	W =    40.518 deg,	P =    40.131 deg,	R =    79.815 deg
   GP2:
	UF : 1, UT : 1,
	J1=    80.000 deg,	J2=    90.000 deg
};
P[269]{
   GP1:
	UF : 1, UT : 1,		CONFIG : 'N U T, 0, 0, 0',
	X =  1902.999  mm,	Y =   -46.261  mm,	Z =   175.051  mm,
	W =    52.365 deg,	P =    -4.474 deg,	R =   -14.021 deg
   GP2:
	UF : 1, UT : 1,
	J1=    90.000 deg,	J2=    90.000 deg
};
P[270]{
   GP1:
	UF : 1, UT : 1,		CONFIG : 'N U T, 0, 0, 0',
	X =  1161.856  mm,	Y =   -92.689  mm,	Z =   175.051  mm,
	W =    38.130 deg,	P =    -5.720 deg,	R =    -4.359 deg
   GP2:
	UF : 1, UT : 1,
	J1=    90.000 deg,	J2=    90.000 deg
};
P[271]{
   GP1:
	UF : 1, UT : 1,		CONFIG : 'N U T, 0, 0, 0',
	X =  1353.427  mm,	Y =   457.025  mm,	Z =   417.051  mm,
	W =    -2.563 deg,	P =     5.520 deg,	R =     2.347 deg
   GP2:
	UF : 1, UT : 1,
	J1=    90.000 deg,	J2=    90.000 deg
};
P[272]{
   GP1:
	UF : 1, UT : 1,		CONFIG : 'N U T, 0, 0, 0',
	X =  1530.428  mm,	Y =   623.025  mm,	Z =   175.051  mm,
	W =   -41.304 deg,	P =     5.776 deg,	R =    -1.616 deg
   GP2:
	UF : 1, UT : 1,
	J1=    90.000 deg,	J2=    90.000 deg
};
P[273]{
   GP1:
	UF : 1, UT : 1,		CONFIG : 'N U T, 0, 0, 0',
	X =  2221.857  mm,	Y =   134.025  mm,	Z =   133.501  mm,
	W =   -39.814 deg,	P =   -13.337 deg,	R =   -23.619 deg
   GP2:
	UF : 1, UT : 1,
	J1=    90.000 deg,	J2=    90.000 deg
};
P[274]{
   GP1:
	UF : 1, UT : 1,		CONFIG : 'N U T, 0, 0, 0',
	X =  1662.172  mm,	Y =  -195.303  mm,	Z =   -14.365  mm,
	W =    38.570 deg,	P =    15.648 deg,	R =    22.724 deg
   GP2:
	UF : 1, UT : 1,
	J1=    90.000 deg,	J2=    90.000 deg
};
P[275]{
   GP1:
	UF : 1, UT : 1,		CONFIG : 'N U T, 0, 0, 0',
	X =  1700.747  mm,	Y =  -196.414  mm,	Z =   -14.295  mm,
	W =    38.571 deg,	P =    15.644 deg,	R =   -27.579 deg
   GP2:
	UF : 1, UT : 1,
	J1=    90.000 deg,	J2=    90.000 deg
};
P[276]{
   GP1:
	UF : 1, UT : 1,		CONFIG : 'N U T, 0, 0, 0',
	X =  2162.665  mm,	Y =   110.242  mm,	Z =    59.358  mm,
	W =   -44.607 deg,	P =    -6.682 deg,	R =    -6.729 deg
   GP2:
	UF : 1, UT : 1,
	J1=    90.000 deg,	J2=    90.000 deg
};
P[277]{
   GP1:
	UF : 1, UT : 1,		CONFIG : 'N U T, 0, 0, 0',
	X =  1967.532  mm,	Y =  -196.842  mm,	Z =   -17.295  mm,
	W =    38.571 deg,	P =    15.644 deg,	R =   -27.579 deg
   GP2:
	UF : 1, UT : 1,
	J1=    90.000 deg,	J2=    90.000 deg
};
P[278]{
   GP1:
	UF : 1, UT : 1,		CONFIG : 'N U T, 0, 0, 0',
	X =  1986.786  mm,	Y =  -196.805  mm,	Z =   -16.016  mm,
	W =    40.162 deg,	P =    14.985 deg,	R =   -66.520 deg
   GP2:
	UF : 1, UT : 1,
	J1=    89.996 deg,	J2=    90.000 deg
};
P[279]{
   GP1:
	UF : 1, UT : 1,		CONFIG : 'N U T, 0, 0, 0',
	X =  2220.705  mm,	Y =    45.955  mm,	Z =    -6.075  mm,
	W =    44.920 deg,	P =     3.025 deg,	R =    -3.029 deg
   GP2:
	UF : 1, UT : 1,
	J1=    90.000 deg,	J2=    90.000 deg
};
P[280]{
   GP1:
	UF : 1, UT : 1,		CONFIG : 'N U T, 0, 0, 0',
	X =  2200.817  mm,	Y =   103.879  mm,	Z =    45.598  mm,
	W =   -44.607 deg,	P =    -6.682 deg,	R =    -6.729 deg
   GP2:
	UF : 1, UT : 1,
	J1=    90.000 deg,	J2=    90.000 deg
};
P[281]{
   GP1:
	UF : 1, UT : 1,		CONFIG : 'N U T, 0, 0, 0',
	X =  1991.025  mm,	Y =   103.879  mm,	Z =    45.598  mm,
	W =   -44.607 deg,	P =    -6.682 deg,	R =    -6.729 deg
   GP2:
	UF : 1, UT : 1,
	J1=    90.000 deg,	J2=    90.000 deg
};
P[282]{
   GP1:
	UF : 1, UT : 1,		CONFIG : 'N U T, 0, 0, 0',
	X =  2256.491  mm,	Y =    45.955  mm,	Z =    -6.075  mm,
	W =    44.920 deg,	P =     3.025 deg,	R =    -3.029 deg
   GP2:
	UF : 1, UT : 1,
	J1=    90.000 deg,	J2=    90.000 deg
};
P[283]{
   GP1:
	UF : 1, UT : 1,		CONFIG : 'N U T, 0, 0, 0',
	X =  2146.075  mm,	Y =    43.814  mm,	Z =   -11.025  mm,
	W =    44.920 deg,	P =     3.025 deg,	R =    -3.029 deg
   GP2:
	UF : 1, UT : 1,
	J1=    90.000 deg,	J2=    90.000 deg
};
P[284]{
   GP1:
	UF : 1, UT : 1,		CONFIG : 'N U T, 0, 0, 0',
	X =  2199.218  mm,	Y =    43.814  mm,	Z =   -11.025  mm,
	W =    44.920 deg,	P =     3.025 deg,	R =    -3.029 deg
   GP2:
	UF : 1, UT : 1,
	J1=    90.000 deg,	J2=    90.000 deg
};
P[285]{
   GP1:
	UF : 1, UT : 1,		CONFIG : 'N U T, 0, 0, 0',
	X =  2086.451  mm,	Y =   114.405  mm,	Z =   133.369  mm,
	W =   -44.606 deg,	P =    -6.682 deg,	R =     6.426 deg
   GP2:
	UF : 1, UT : 1,
	J1=    90.000 deg,	J2=    90.000 deg
};
P[286]{
   GP1:
	UF : 1, UT : 1,		CONFIG : 'N U T, 0, 0, 0',
	X =  2121.394  mm,	Y =   114.404  mm,	Z =   147.283  mm,
	W =   -41.424 deg,	P =   -19.434 deg,	R =   -97.506 deg
   GP2:
	UF : 1, UT : 1,
	J1=    90.000 deg,	J2=   100.000 deg
};
P[287]{
   GP1:
	UF : 1, UT : 1,		CONFIG : 'N U T, 0, 0, 0',
	X =  2080.531  mm,	Y =    -7.596  mm,	Z =    92.282  mm,
	W =   -41.424 deg,	P =   -19.434 deg,	R =   -97.506 deg
   GP2:
	UF : 1, UT : 1,
	J1=    90.000 deg,	J2=   100.000 deg
};
P[288]{
   GP1:
	UF : 1, UT : 1,		CONFIG : 'N U T, 0, 0, 0',
	X =  2206.218  mm,	Y =    43.813  mm,	Z =   -11.025  mm,
	W =    44.920 deg,	P =     3.025 deg,	R =   -14.671 deg
   GP2:
	UF : 1, UT : 1,
	J1=    90.000 deg,	J2=    90.000 deg
};
P[289]{
   GP1:
	UF : 1, UT : 1,		CONFIG : 'N U T, 0, 0, 0',
	X =  2110.963  mm,	Y =    44.118  mm,	Z =   -20.037  mm,
	W =    44.927 deg,	P =     3.029 deg,	R =     5.583 deg
   GP2:
	UF : 1, UT : 1,
	J1=    90.000 deg,	J2=    90.000 deg
};
P[290]{
   GP1:
	UF : 1, UT : 1,		CONFIG : 'N U T, 0, 0, 0',
	X =  2080.530  mm,	Y =    -7.596  mm,	Z =    92.282  mm,
	W =   -41.424 deg,	P =   -19.434 deg,	R =   -97.506 deg
   GP2:
	UF : 1, UT : 1,
	J1=    90.000 deg,	J2=   100.000 deg
};
P[291]{
   GP1:
	UF : 1, UT : 1,		CONFIG : 'N U T, 0, 0, 0',
	X =  2080.530  mm,	Y =   309.547  mm,	Z =   503.711  mm,
	W =    -3.830 deg,	P =   -10.878 deg,	R =   -17.892 deg
   GP2:
	UF : 1, UT : 1,
	J1=    90.000 deg,	J2=   135.000 deg
};
P[292]{
   GP1:
	UF : 1, UT : 1,		CONFIG : 'N U T, 0, 0, 0',
	X =  2670.559  mm,	Y =   209.547  mm,	Z =   314.711  mm,
	W =    -3.830 deg,	P =   -10.878 deg,	R =   -17.892 deg
   GP2:
	UF : 1, UT : 1,
	J1=    90.000 deg,	J2=   135.000 deg
};
P[293]{
   GP1:
	UF : 1, UT : 1,		CONFIG : 'N U T, 0, 0, 0',
	X =  2021.034  mm,	Y =    44.118  mm,	Z =   -20.036  mm,
	W =    44.927 deg,	P =     3.029 deg,	R =     5.583 deg
   GP2:
	UF : 1, UT : 1,
	J1=    90.000 deg,	J2=    90.000 deg
};
P[294]{
   GP1:
	UF : 1, UT : 1,		CONFIG : 'N U T, 0, 0, 0',
	X =  2006.091  mm,	Y =    44.761  mm,	Z =   -20.036  mm,
	W =    44.926 deg,	P =     3.029 deg,	R =    37.260 deg
   GP2:
	UF : 1, UT : 1,
	J1=    90.000 deg,	J2=    90.000 deg
};
P[295]{
   GP1:
	UF : 1, UT : 1,		CONFIG : 'N U T, 0, 0, 0',
	X =  2649.168  mm,	Y =   166.049  mm,	Z =   301.659  mm,
	W =    13.374 deg,	P =   -35.036 deg,	R =   -22.495 deg
   GP2:
	UF : 1, UT : 1,
	J1=    90.000 deg,	J2=   135.000 deg
};
P[296]{
   GP1:
	UF : 1, UT : 1,		CONFIG : 'N U T, 0, 0, 0',
	X =  2349.168  mm,	Y =   281.049  mm,	Z =   301.659  mm,
	W =     -.090 deg,	P =    -5.498 deg,	R =      .950 deg
   GP2:
	UF : 1, UT : 1,
	J1=    90.000 deg,	J2=   135.000 deg
};
P[297]{
   GP1:
	UF : 1, UT : 1,		CONFIG : 'N U T, 0, 0, 0',
	X =  1789.966  mm,	Y =    44.323  mm,	Z =    52.714  mm,
	W =    50.325 deg,	P =     2.535 deg,	R =    12.049 deg
   GP2:
	UF : 1, UT : 1,
	J1=    90.000 deg,	J2=    90.000 deg
};
P[298]{
   GP1:
	UF : 1, UT : 1,		CONFIG : 'N U T, 0, 0, 0',
	X =  1683.323  mm,	Y =    44.322  mm,	Z =    52.714  mm,
	W =    50.813 deg,	P =     2.431 deg,	R =    12.070 deg
   GP2:
	UF : 1, UT : 1,
	J1=    90.000 deg,	J2=    90.000 deg
};
P[299]{
   GP1:
	UF : 1, UT : 1,		CONFIG : 'N U T, 0, 0, 0',
	X =  2703.820  mm,	Y =   252.204  mm,	Z =   224.219  mm,
	W =     -.140 deg,	P =    -8.465 deg,	R =      .956 deg
   GP2:
	UF : 1, UT : 1,
	J1=    90.000 deg,	J2=   135.000 deg
};
P[300]{
   GP1:
	UF : 1, UT : 1,		CONFIG : 'N U T, 0, 0, 0',
	X =  2289.178  mm,	Y =   268.490  mm,	Z =   224.220  mm,
	W =     -.140 deg,	P =    -8.465 deg,	R =      .956 deg
   GP2:
	UF : 1, UT : 1,
	J1=    90.000 deg,	J2=   135.000 deg
};
P[301]{
   GP1:
	UF : 1, UT : 1,		CONFIG : 'N U T, 0, 0, 0',
	X =  1843.464  mm,	Y =   431.347  mm,	Z =   609.934  mm,
	W =     -.140 deg,	P =    -8.465 deg,	R =   -19.002 deg
   GP2:
	UF : 1, UT : 1,
	J1=    90.000 deg,	J2=   135.000 deg
};
P[302]{
   GP1:
	UF : 1, UT : 1,		CONFIG : 'N U T, 0, 0, 0',
	X =  1843.464  mm,	Y =   431.347  mm,	Z =   378.506  mm,
	W =    39.110 deg,	P =     2.688 deg,	R =   -82.797 deg
   GP2:
	UF : 1, UT : 1,
	J1=    90.000 deg,	J2=    90.000 deg
};
P[303]{
   GP1:
	UF : 1, UT : 1,		CONFIG : 'N U T, 0, 0, 0',
	X =  2020.464  mm,	Y =   107.456  mm,	Z =   101.505  mm,
	W =    39.110 deg,	P =     2.688 deg,	R =   -82.797 deg
   GP2:
	UF : 1, UT : 1,
	J1=    90.000 deg,	J2=    90.000 deg
};
P[304]{
   GP1:
	UF : 1, UT : 1,		CONFIG : 'N U T, 0, 0, 0',
	X =  1667.771  mm,	Y =    42.806  mm,	Z =    54.038  mm,
	W =    53.172 deg,	P =     1.611 deg,	R =    24.177 deg
   GP2:
	UF : 1, UT : 1,
	J1=    90.000 deg,	J2=    90.000 deg
};
P[305]{
   GP1:
	UF : 1, UT : 1,		CONFIG : 'N U T, 0, 0, 0',
	X =  1826.870  mm,	Y =    43.892  mm,	Z =    52.359  mm,
	W =    53.726 deg,	P =    -4.474 deg,	R =     3.443 deg
   GP2:
	UF : 1, UT : 1,
	J1=    90.000 deg,	J2=    90.000 deg
};
P[306]{
   GP1:
	UF : 1, UT : 1,		CONFIG : 'N U T, 0, 0, 0',
	X =  1963.585  mm,	Y =    45.392  mm,	Z =    50.646  mm,
	W =    53.726 deg,	P =    -4.474 deg,	R =     3.443 deg
   GP2:
	UF : 1, UT : 1,
	J1=    90.000 deg,	J2=    90.000 deg
};
P[307]{
   GP1:
	UF : 1, UT : 1,		CONFIG : 'N U T, 0, 0, -1',
	X =  2012.815  mm,	Y =   114.104  mm,	Z =    90.700  mm,
	W =    40.362 deg,	P =    21.867 deg,	R =  -139.995 deg
   GP2:
	UF : 1, UT : 1,
	J1=    90.000 deg,	J2=    90.000 deg
};
P[308]{
   GP1:
	UF : 1, UT : 1,		CONFIG : 'N U T, 0, 0, 0',
	X =  1644.243  mm,	Y =   456.961  mm,	Z =    90.700  mm,
	W =   -42.959 deg,	P =    14.926 deg,	R =    16.534 deg
   GP2:
	UF : 1, UT : 1,
	J1=    90.000 deg,	J2=    90.000 deg
};
P[309]{
   GP1:
	UF : 1, UT : 1,		CONFIG : 'N U T, 0, 0, 0',
	X =  1667.302  mm,	Y =   122.961  mm,	Z =    90.700  mm,
	W =   -42.959 deg,	P =    14.926 deg,	R =    16.534 deg
   GP2:
	UF : 1, UT : 1,
	J1=    90.000 deg,	J2=    90.000 deg
};
P[310]{
   GP1:
	UF : 1, UT : 1,		CONFIG : 'N U T, 0, 0, 0',
	X =  1987.759  mm,	Y =    40.243  mm,	Z =    54.128  mm,
	W =    53.726 deg,	P =    -4.474 deg,	R =   -26.684 deg
   GP2:
	UF : 1, UT : 1,
	J1=    90.000 deg,	J2=    90.000 deg
};
P[311]{
   GP1:
	UF : 1, UT : 1,		CONFIG : 'N U T, 0, 0, 0',
	X =  2224.159  mm,	Y =    58.556  mm,	Z =    -5.448  mm,
	W =   -44.607 deg,	P =    -6.682 deg,	R =    -6.729 deg
   GP2:
	UF : 1, UT : 1,
	J1=    90.000 deg,	J2=    90.000 deg
};
P[312]{
   GP1:
	UF : 1, UT : 1,		CONFIG : 'N U T, 0, 0, 0',
	X =  2258.659  mm,	Y =    57.913  mm,	Z =    -5.448  mm,
	W =   -44.607 deg,	P =    -6.682 deg,	R =    -6.729 deg
   GP2:
	UF : 1, UT : 1,
	J1=    90.000 deg,	J2=    90.000 deg
};
P[313]{
   GP1:
	UF : 1, UT : 1,		CONFIG : 'N U T, 0, 0, 0',
	X =  2132.012  mm,	Y =    56.491  mm,	Z =   -12.327  mm,
	W =   -44.606 deg,	P =    -6.681 deg,	R =    -6.729 deg
   GP2:
	UF : 1, UT : 1,
	J1=    90.000 deg,	J2=    90.000 deg
};
P[314]{
   GP1:
	UF : 1, UT : 1,		CONFIG : 'N U T, 0, 0, 0',
	X =  2200.013  mm,	Y =    57.134  mm,	Z =   -12.327  mm,
	W =   -44.606 deg,	P =    -6.681 deg,	R =    -6.729 deg
   GP2:
	UF : 1, UT : 1,
	J1=    90.000 deg,	J2=    90.000 deg
};
P[315]{
   GP1:
	UF : 1, UT : 1,		CONFIG : 'N U T, 0, 0, 0',
	X =  2209.513  mm,	Y =    57.348  mm,	Z =   -12.326  mm,
	W =   -44.606 deg,	P =    -6.681 deg,	R =     3.931 deg
   GP2:
	UF : 1, UT : 1,
	J1=    90.000 deg,	J2=    90.000 deg
};
P[316]{
   GP1:
	UF : 1, UT : 1,		CONFIG : 'N U T, 0, 0, 0',
	X =  1985.356  mm,	Y =    56.787  mm,	Z =   -20.825  mm,
	W =   -44.607 deg,	P =    -6.682 deg,	R =    -3.024 deg
   GP2:
	UF : 1, UT : 1,
	J1=    90.000 deg,	J2=    90.000 deg
};
P[317]{
   GP1:
	UF : 1, UT : 1,		CONFIG : 'N U T, 0, 0, 0',
	X =  2092.498  mm,	Y =    57.858  mm,	Z =   -20.825  mm,
	W =   -44.607 deg,	P =    -6.682 deg,	R =    -3.024 deg
   GP2:
	UF : 1, UT : 1,
	J1=    90.000 deg,	J2=    90.000 deg
};
P[318]{
   GP1:
	UF : 1, UT : 1,		CONFIG : 'N U T, 0, 0, 0',
	X =  2108.090  mm,	Y =    59.550  mm,	Z =   -18.097  mm,
	W =   -41.242 deg,	P =   -19.883 deg,	R =    20.906 deg
   GP2:
	UF : 1, UT : 1,
	J1=    90.000 deg,	J2=    90.000 deg
};
P[319]{
   GP1:
	UF : 1, UT : 1,		CONFIG : 'N U T, 0, 0, 0',
	X =  2003.979  mm,	Y =    88.747  mm,	Z =   -10.736  mm,
	W =   -45.251 deg,	P =    -8.450 deg,	R =  -108.138 deg
   GP2:
	UF : 1, UT : 1,
	J1=    90.000 deg,	J2=   100.000 deg
};
P[320]{
   GP1:
	UF : 1, UT : 1,		CONFIG : 'N U T, 0, 0, 0',
	X =  2002.512  mm,	Y =  -133.508  mm,	Z =   -48.404  mm,
	W =   -45.251 deg,	P =    -8.450 deg,	R =   -86.327 deg
   GP2:
	UF : 1, UT : 1,
	J1=    90.000 deg,	J2=   100.000 deg
};
P[321]{
   GP1:
	UF : 1, UT : 1,		CONFIG : 'N U T, 0, 0, 0',
	X =  1385.322  mm,	Y =    99.987  mm,	Z =    81.524  mm,
	W =   -41.156 deg,	P =    19.919 deg,	R =    36.091 deg
   GP2:
	UF : 1, UT : 1,
	J1=    90.000 deg,	J2=    90.000 deg
};
P[322]{
   GP1:
	UF : 1, UT : 1,		CONFIG : 'N U T, 0, 0, 0',
	X =  1287.575  mm,	Y =   726.729  mm,	Z =   436.468  mm,
	W =   -45.215 deg,	P =    11.103 deg,	R =    59.860 deg
   GP2:
	UF : 1, UT : 1,
	J1=    90.000 deg,	J2=    90.000 deg
};
P[323]{
   GP1:
	UF : 1, UT : 1,		CONFIG : 'N U T, 0, 0, 0',
	X =  2772.800  mm,	Y =  1353.842  mm,	Z =    52.554  mm,
	W =      .247 deg,	P =     2.267 deg,	R =    25.456 deg
   GP2:
	UF : 1, UT : 1,
	J1=    90.000 deg,	J2=    90.000 deg
};
P[324]{
   GP1:
	UF : 1, UT : 1,		CONFIG : 'N U T, 0, 0, 0',
	X =  2849.615  mm,	Y =  1373.219  mm,	Z =     2.246  mm,
	W =      .303 deg,	P =     1.056 deg,	R =    25.442 deg
   GP2:
	UF : 1, UT : 1,
	J1=    89.998 deg,	J2=    90.000 deg
};
P[325]{
   GP1:
	UF : 1, UT : 1,		CONFIG : 'N U B, 0, 0, 0',
	X =   356.032  mm,	Y =    -2.146  mm,	Z =  2424.049  mm,
	W =      .001 deg,	P =   -40.002 deg,	R =     -.005 deg
   GP2:
	UF : 1, UT : 1,
	J1=   -90.000 deg,	J2=    90.000 deg
};
P[326]{
   GP1:
	UF : 1, UT : 1,		CONFIG : 'N U T, 0, 0, 0',
	X =  1109.146  mm,	Y =  -695.879  mm,	Z =  1059.006  mm,
	W =   -45.665 deg,	P =    -3.656 deg,	R =    28.137 deg
   GP2:
	UF : 1, UT : 1,
	J1=   -90.000 deg,	J2=    90.000 deg
};
P[327]{
   GP1:
	UF : 1, UT : 1,		CONFIG : 'N U T, 0, 0, 0',
	X =  2182.795  mm,	Y =   -54.409  mm,	Z =  -297.620  mm,
	W =    -4.848 deg,	P =     4.640 deg,	R =    10.727 deg
   GP2:
	UF : 1, UT : 1,
	J1=    45.000 deg,	J2=   182.246 deg
};
P[328]{
   GP1:
	UF : 1, UT : 1,		CONFIG : 'N U T, 0, 0, 0',
	X =  2785.854  mm,	Y =  1360.233  mm,	Z =    51.016  mm,
	W =      .260 deg,	P =     1.052 deg,	R =    25.457 deg
   GP2:
	UF : 1, UT : 1,
	J1=    90.000 deg,	J2=    90.000 deg
};
P[329]{
   GP1:
	UF : 1, UT : 1,		CONFIG : 'N U T, 0, 0, 0',
	X =  1254.943  mm,	Y =   301.685  mm,	Z =   234.946  mm,
	W =   -61.903 deg,	P =    47.077 deg,	R =    68.180 deg
   GP2:
	UF : 1, UT : 1,
	J1=    90.000 deg,	J2=    90.000 deg
};
P[330]{
   GP1:
	UF : 1, UT : 1,		CONFIG : 'N U T, 0, 0, 0',
	X =  2415.039  mm,	Y =   -85.100  mm,	Z =   -32.227  mm,
	W =   -21.721 deg,	P =   -27.900 deg,	R =   -19.487 deg
   GP2:
	UF : 1, UT : 1,
	J1=    90.000 deg,	J2=   100.000 deg
};
P[331]{
   GP1:
	UF : 1, UT : 1,		CONFIG : 'N U T, 0, 0, 0',
	X =  1217.104  mm,	Y =  -169.780  mm,	Z =   187.729  mm,
	W =   -34.745 deg,	P =    30.619 deg,	R =   119.475 deg
   GP2:
	UF : 1, UT : 1,
	J1=    90.000 deg,	J2=    90.000 deg
};
P[332]{
   GP1:
	UF : 1, UT : 1,		CONFIG : 'N U T, 0, 0, 0',
	X =  1573.104  mm,	Y =  -218.075  mm,	Z =    59.729  mm,
	W =   -34.744 deg,	P =    30.618 deg,	R =   128.397 deg
   GP2:
	UF : 1, UT : 1,
	J1=    90.000 deg,	J2=    90.000 deg
};
P[333]{
   GP1:
	UF : 1, UT : 1,		CONFIG : 'N U T, 0, 0, 0',
	X =  2754.450  mm,	Y =   160.116  mm,	Z =   172.316  mm,
	W =     2.791 deg,	P =    -7.674 deg,	R =   -18.462 deg
   GP2:
	UF : 1, UT : 1,
	J1=    90.000 deg,	J2=   135.000 deg
};
P[334]{
   GP1:
	UF : 1, UT : 1,		CONFIG : 'N U T, 0, 0, 0',
	X =  2866.212  mm,	Y =   161.367  mm,	Z =   172.734  mm,
	W =     9.505 deg,	P =   -26.592 deg,	R =   -20.508 deg
   GP2:
	UF : 1, UT : 1,
	J1=    90.000 deg,	J2=   135.000 deg
};
P[335]{
   GP1:
	UF : 1, UT : 1,		CONFIG : 'N U T, 0, 0, 1',
	X =  1459.008  mm,	Y =   -74.800  mm,	Z =   199.820  mm,
	W =   -34.742 deg,	P =    30.617 deg,	R =   153.799 deg
   GP2:
	UF : 1, UT : 1,
	J1=    90.000 deg,	J2=    90.000 deg
};
P[336]{
   GP1:
	UF : 1, UT : 1,		CONFIG : 'N U T, 0, 0, 0',
	X =  1319.009  mm,	Y =  -291.799  mm,	Z =   199.820  mm,
	W =    44.863 deg,	P =    -3.871 deg,	R =     -.364 deg
   GP2:
	UF : 1, UT : 1,
	J1=    90.000 deg,	J2=    90.000 deg
};
P[337]{
   GP1:
	UF : 1, UT : 1,		CONFIG : 'N U T, 0, 0, 0',
	X =  2390.009  mm,	Y =  -240.799  mm,	Z =    52.820  mm,
	W =    42.099 deg,	P =    -2.376 deg,	R =   -15.667 deg
   GP2:
	UF : 1, UT : 1,
	J1=    90.000 deg,	J2=    90.000 deg
};
P[338]{
   GP1:
	UF : 1, UT : 1,		CONFIG : 'N U T, 0, 0, 0',
	X =  2377.770  mm,	Y =   263.073  mm,	Z =    82.894  mm,
	W =     1.905 deg,	P =     -.030 deg,	R =      .945 deg
   GP2:
	UF : 1, UT : 1,
	J1=    90.000 deg,	J2=   135.000 deg
};
P[339]{
   GP1:
	UF : 1, UT : 1,		CONFIG : 'N U T, 0, 0, 0',
	X =  2746.516  mm,	Y =   264.236  mm,	Z =    82.888  mm,
	W =     2.767 deg,	P =     -.044 deg,	R =      .944 deg
   GP2:
	UF : 1, UT : 1,
	J1=    90.000 deg,	J2=   135.000 deg
};
P[340]{
   GP1:
	UF : 1, UT : 1,		CONFIG : 'N U T, 0, 0, 0',
	X =  2502.492  mm,	Y =  -211.230  mm,	Z =    67.973  mm,
	W =    44.580 deg,	P =     6.891 deg,	R =   -21.154 deg
   GP2:
	UF : 1, UT : 1,
	J1=    90.000 deg,	J2=    90.000 deg
};
P[341]{
   GP1:
	UF : 1, UT : 1,		CONFIG : 'N U T, 0, 0, 0',
	X =  2329.524  mm,	Y =  -211.230  mm,	Z =    67.973  mm,
	W =    44.580 deg,	P =     6.891 deg,	R =   -21.154 deg
   GP2:
	UF : 1, UT : 1,
	J1=    90.000 deg,	J2=    90.000 deg
};
P[342]{
   GP1:
	UF : 1, UT : 1,		CONFIG : 'N U T, 0, 0, 0',
	X =  2329.524  mm,	Y =  -124.230  mm,	Z =    67.973  mm,
	W =    44.580 deg,	P =     6.891 deg,	R =   -21.154 deg
   GP2:
	UF : 1, UT : 1,
	J1=    90.000 deg,	J2=    90.000 deg
};
P[343]{
   GP1:
	UF : 1, UT : 1,		CONFIG : 'N U T, 0, 0, 0',
	X =  2064.146  mm,	Y =   104.765  mm,	Z =   -17.011  mm,
	W =    40.363 deg,	P =    21.868 deg,	R =  -105.672 deg
   GP2:
	UF : 1, UT : 1,
	J1=    90.000 deg,	J2=    90.000 deg
};
P[344]{
   GP1:
	UF : 1, UT : 1,		CONFIG : 'N U T, 0, 0, 0',
	X =  2090.504  mm,	Y =    81.118  mm,	Z =   -17.883  mm,
	W =    40.363 deg,	P =    21.868 deg,	R =  -105.672 deg
   GP2:
	UF : 1, UT : 1,
	J1=    90.000 deg,	J2=    90.000 deg
};
P[345]{
   GP1:
	UF : 1, UT : 1,		CONFIG : 'N U T, 0, 0, -1',
	X =  2109.088  mm,	Y =    63.501  mm,	Z =   -16.040  mm,
	W =    40.363 deg,	P =    21.868 deg,	R =  -130.780 deg
   GP2:
	UF : 1, UT : 1,
	J1=    90.000 deg,	J2=    90.000 deg
};
P[346]{
   GP1:
	UF : 1, UT : 1,		CONFIG : 'N U T, 0, 0, 0',
	X =  2329.524  mm,	Y =  -124.230  mm,	Z =    67.973  mm,
	W =    44.580 deg,	P =     6.891 deg,	R =   -21.154 deg
   GP2:
	UF : 1, UT : 1,
	J1=    90.000 deg,	J2=    90.000 deg
};
P[347]{
   GP1:
	UF : 1, UT : 1,		CONFIG : 'N U T, 0, 0, 0',
	X =  1069.524  mm,	Y =  -124.230  mm,	Z =   124.973  mm,
	W =    53.137 deg,	P =    27.952 deg,	R =    15.270 deg
   GP2:
	UF : 1, UT : 1,
	J1=    90.000 deg,	J2=    90.000 deg
};
P[348]{
   GP1:
	UF : 1, UT : 1,		CONFIG : 'N U T, 0, 0, 0',
	X =  1062.033  mm,	Y =   -72.059  mm,	Z =  1104.020  mm,
	W =     1.209 deg,	P =    20.107 deg,	R =    63.832 deg
   GP2:
	UF : 1, UT : 1,
	J1=    90.000 deg,	J2=    90.000 deg
};
P[349]{
   GP1:
	UF : 1, UT : 1,		CONFIG : 'N U T, 0, 0, 0',
	X =  1214.600  mm,	Y =   479.028  mm,	Z =   916.465  mm,
	W =    39.867 deg,	P =   -22.888 deg,	R =   -38.695 deg
   GP2:
	UF : 1, UT : 1,
	J1=   -90.000 deg,	J2=   -90.000 deg
};
P[350]{
   GP1:
	UF : 1, UT : 1,		CONFIG : 'N U T, 0, 0, 0',
	X =   713.970  mm,	Y =   812.888  mm,	Z =  1598.123  mm,
	W =    60.754 deg,	P =   -26.996 deg,	R =   -17.604 deg
   GP2:
	UF : 1, UT : 1,
	J1=   -90.000 deg,	J2=   -90.000 deg
};
P[351]{
   GP1:
	UF : 1, UT : 1,		CONFIG : 'N U T, 0, 0, 0',
	X =  1615.600  mm,	Y =   479.028  mm,	Z =   916.465  mm,
	W =    39.867 deg,	P =   -22.888 deg,	R =   -65.014 deg
   GP2:
	UF : 1, UT : 1,
	J1=   -90.000 deg,	J2=   -90.000 deg
};
P[352]{
   GP1:
	UF : 1, UT : 1,		CONFIG : 'N U T, 0, 0, 0',
	X =  1684.217  mm,	Y =    62.865  mm,	Z =   -15.611  mm,
	W =   -42.812 deg,	P =    15.443 deg,	R =    16.036 deg
   GP2:
	UF : 1, UT : 1,
	J1=    90.000 deg,	J2=    90.000 deg
};
P[353]{
   GP1:
	UF : 1, UT : 1,		CONFIG : 'N U T, 0, 0, 0',
	X =  1641.653  mm,	Y =    60.501  mm,	Z =   -17.464  mm,
	W =   -42.812 deg,	P =    15.444 deg,	R =    16.036 deg
   GP2:
	UF : 1, UT : 1,
	J1=    90.000 deg,	J2=    90.000 deg
};
P[354]{
   GP1:
	UF : 1, UT : 1,		CONFIG : 'N U T, 0, 0, 0',
	X =  1637.009  mm,	Y =    61.569  mm,	Z =   -16.757  mm,
	W =   -42.812 deg,	P =    15.443 deg,	R =    -7.967 deg
   GP2:
	UF : 1, UT : 1,
	J1=    90.000 deg,	J2=    90.000 deg
};
P[355]{
   GP1:
	UF : 1, UT : 1,		CONFIG : 'N U T, 0, 0, 0',
	X =  1629.863  mm,	Y =    63.510  mm,	Z =   -19.559  mm,
	W =   -38.593 deg,	P =    25.218 deg,	R =   -16.905 deg
   GP2:
	UF : 1, UT : 1,
	J1=    90.000 deg,	J2=    90.000 deg
};
P[356]{
   GP1:
	UF : 1, UT : 1,		CONFIG : 'N U T, 0, 0, 0',
	X =  1602.812  mm,	Y =    92.790  mm,	Z =   -18.625  mm,
	W =   -38.593 deg,	P =    25.219 deg,	R =   -16.905 deg
   GP2:
	UF : 1, UT : 1,
	J1=    90.000 deg,	J2=    90.000 deg
};
P[357]{
   GP1:
	UF : 1, UT : 1,		CONFIG : 'N U T, 0, 0, 0',
	X =  1580.378  mm,	Y =   103.834  mm,	Z =   -17.928  mm,
	W =   -47.725 deg,	P =    -3.150 deg,	R =      .571 deg
   GP2:
	UF : 1, UT : 1,
	J1=    90.000 deg,	J2=    90.000 deg
};
P[358]{
   GP1:
	UF : 1, UT : 1,		CONFIG : 'N U T, 0, 0, 0',
	X =  1552.243  mm,	Y =    77.783  mm,	Z =   -20.604  mm,
	W =   -41.216 deg,	P =    19.944 deg,	R =    98.982 deg
   GP2:
	UF : 1, UT : 1,
	J1=    90.000 deg,	J2=    90.000 deg
};
P[359]{
   GP1:
	UF : 1, UT : 1,		CONFIG : 'N U T, 0, 0, 0',
	X =  1548.399  mm,	Y =    36.103  mm,	Z =   -14.087  mm,
	W =   -41.216 deg,	P =    19.935 deg,	R =    99.346 deg
   GP2:
	UF : 1, UT : 1,
	J1=    89.998 deg,	J2=    90.000 deg
};
P[360]{
   GP1:
	UF : 1, UT : 1,		CONFIG : 'N U T, 0, 0, 0',
	X =  1704.637  mm,	Y =   898.337  mm,	Z =  1001.782  mm,
	W =   -20.210 deg,	P =   -41.106 deg,	R =     1.246 deg
   GP2:
	UF : 1, UT : 1,
	J1=   -90.000 deg,	J2=   -90.000 deg
};
P[361]{
   GP1:
	UF : 1, UT : 1,		CONFIG : 'N U T, 0, 0, 0',
	X =  1682.137  mm,	Y =   345.195  mm,	Z =   941.171  mm,
	W =    42.022 deg,	P =   -15.891 deg,	R =   -33.571 deg
   GP2:
	UF : 1, UT : 1,
	J1=   -90.000 deg,	J2=   -90.000 deg
};
P[362]{
   GP1:
	UF : 1, UT : 1,		CONFIG : 'N U T, 0, 0, 0',
	X =  1546.344  mm,	Y =    26.267  mm,	Z =   -13.494  mm,
	W =   -41.215 deg,	P =    19.944 deg,	R =    68.893 deg
   GP2:
	UF : 1, UT : 1,
	J1=    89.999 deg,	J2=    90.000 deg
};
P[363]{
   GP1:
	UF : 1, UT : 1,		CONFIG : 'N U T, 0, 0, 0',
	X =  1542.801  mm,	Y =    22.402  mm,	Z =   -15.264  mm,
	W =   -41.215 deg,	P =    19.944 deg,	R =    32.568 deg
   GP2:
	UF : 1, UT : 1,
	J1=    90.000 deg,	J2=    90.000 deg
};
P[364]{
   GP1:
	UF : 1, UT : 1,		CONFIG : 'N U T, 0, 0, 0',
	X =  1535.086  mm,	Y =    20.188  mm,	Z =   -15.264  mm,
	W =   -41.215 deg,	P =    19.944 deg,	R =    32.568 deg
   GP2:
	UF : 1, UT : 1,
	J1=    90.000 deg,	J2=    90.000 deg
};
P[365]{
   GP1:
	UF : 1, UT : 1,		CONFIG : 'N U T, 0, 0, 0',
	X =  2357.041  mm,	Y =   -23.041  mm,	Z =    82.290  mm,
	W =   -26.718 deg,	P =   -22.770 deg,	R =   -10.639 deg
   GP2:
	UF : 1, UT : 1,
	J1=    90.000 deg,	J2=   100.000 deg
};
P[366]{
   GP1:
	UF : 1, UT : 1,		CONFIG : 'N U T, 0, 0, 0',
	X =  2407.215  mm,	Y =    96.473  mm,	Z =   834.886  mm,
	W =     5.388 deg,	P =    42.666 deg,	R =    25.064 deg
   GP2:
	UF : 1, UT : 1,
	J1=    89.999 deg,	J2=   -90.000 deg
};
P[367]{
   GP1:
	UF : 1, UT : 1,		CONFIG : 'N U T, 0, 0, 0',
	X =  1855.998  mm,	Y =   173.909  mm,	Z =   960.367  mm,
	W =    58.350 deg,	P =   -26.173 deg,	R =   -73.280 deg
   GP2:
	UF : 1, UT : 1,
	J1=   -90.000 deg,	J2=   -90.000 deg
};
P[368]{
   GP1:
	UF : 1, UT : 1,		CONFIG : 'N U T, 0, 0, 0',
	X =  1291.698  mm,	Y =   195.066  mm,	Z =   960.367  mm,
	W =    58.350 deg,	P =   -26.173 deg,	R =   -73.280 deg
   GP2:
	UF : 1, UT : 1,
	J1=   -90.000 deg,	J2=   -90.000 deg
};
P[369]{
   GP1:
	UF : 1, UT : 1,		CONFIG : 'N U T, 0, 0, 1',
	X =  1641.151  mm,	Y =  -211.306  mm,	Z =   -12.671  mm,
	W =   -31.822 deg,	P =    29.963 deg,	R =   131.853 deg
   GP2:
	UF : 1, UT : 1,
	J1=    89.989 deg,	J2=    90.000 deg
};
P[370]{
   GP1:
	UF : 1, UT : 1,		CONFIG : 'N U T, 0, 0, 1',
	X =  1642.822  mm,	Y =    21.416  mm,	Z =   -14.476  mm,
	W =   -34.233 deg,	P =    30.069 deg,	R =   141.356 deg
   GP2:
	UF : 1, UT : 1,
	J1=    90.000 deg,	J2=    90.000 deg
};
P[371]{
   GP1:
	UF : 1, UT : 1,		CONFIG : 'N U T, 0, 0, 0',
	X =  1433.073  mm,	Y =  -528.643  mm,	Z =   576.275  mm,
	W =    -5.611 deg,	P =   -10.020 deg,	R =     8.093 deg
   GP2:
	UF : 1, UT : 1,
	J1=    90.000 deg,	J2=  -100.000 deg
};
P[372]{
   GP1:
	UF : 1, UT : 1,		CONFIG : 'N U T, 0, 0, 0',
	X =  1558.148  mm,	Y =   135.723  mm,	Z =   206.394  mm,
	W =   -46.360 deg,	P =    11.199 deg,	R =    10.858 deg
   GP2:
	UF : 1, UT : 1,
	J1=    90.000 deg,	J2=   -90.000 deg
};
P[373]{
   GP1:
	UF : 1, UT : 1,		CONFIG : 'N U T, 0, 0, 0',
	X =  2022.992  mm,	Y =   -45.728  mm,	Z =     2.837  mm,
	W =   -43.918 deg,	P =    -5.993 deg,	R =   -30.730 deg
   GP2:
	UF : 1, UT : 1,
	J1=    90.000 deg,	J2=   -90.000 deg
};
P[374]{
   GP1:
	UF : 1, UT : 1,		CONFIG : 'N U T, 0, 0, 0',
	X =  2345.985  mm,	Y =  -176.107  mm,	Z =   -12.260  mm,
	W =    44.581 deg,	P =     6.891 deg,	R =    -6.941 deg
   GP2:
	UF : 1, UT : 1,
	J1=    90.000 deg,	J2=    90.000 deg
};
P[375]{
   GP1:
	UF : 1, UT : 1,		CONFIG : 'N U T, 0, 0, 0',
	X =  2520.065  mm,	Y =  -178.161  mm,	Z =   -10.410  mm,
	W =    44.582 deg,	P =     6.891 deg,	R =    -6.941 deg
   GP2:
	UF : 1, UT : 1,
	J1=    90.000 deg,	J2=    90.000 deg
};
P[376]{
   GP1:
	UF : 1, UT : 1,		CONFIG : 'N U T, 0, 0, 0',
	X =  2053.353  mm,	Y =   209.744  mm,	Z =   328.977  mm,
	W =   -44.718 deg,	P =   -17.447 deg,	R =    -6.431 deg
   GP2:
	UF : 1, UT : 1,
	J1=    90.000 deg,	J2=   100.000 deg
};
P[377]{
   GP1:
	UF : 1, UT : 1,		CONFIG : 'N U T, 0, 0, 0',
	X =  1074.532  mm,	Y =  -506.968  mm,	Z =  1238.459  mm,
	W =     -.673 deg,	P =   -46.105 deg,	R =     9.949 deg
   GP2:
	UF : 1, UT : 1,
	J1=   -90.000 deg,	J2=    90.000 deg
};
P[378]{
   GP1:
	UF : 1, UT : 1,		CONFIG : 'N U T, 0, 0, 0',
	X =  1359.532  mm,	Y =  -506.968  mm,	Z =   962.459  mm,
	W =     -.673 deg,	P =   -46.105 deg,	R =     9.949 deg
   GP2:
	UF : 1, UT : 1,
	J1=   -90.000 deg,	J2=    90.000 deg
};
P[379]{
   GP1:
	UF : 1, UT : 1,		CONFIG : 'N U T, 0, 0, 0',
	X =  1645.943  mm,	Y =  -472.973  mm,	Z =   885.320  mm,
	W =   -29.059 deg,	P =   -38.116 deg,	R =    41.980 deg
   GP2:
	UF : 1, UT : 1,
	J1=   -90.000 deg,	J2=    90.000 deg
};
P[380]{
   GP1:
	UF : 1, UT : 1,		CONFIG : 'N U T, 0, 0, 0',
	X =  1214.623  mm,	Y =   483.357  mm,	Z =   914.016  mm,
	W =   -25.369 deg,	P =    11.963 deg,	R =   -19.314 deg
   GP2:
	UF : 1, UT : 1,
	J1=    90.000 deg,	J2=   100.000 deg
};
P[381]{
   GP1:
	UF : 1, UT : 1,		CONFIG : 'N U T, 0, 0, -1',
	X =  1626.194  mm,	Y =   455.887  mm,	Z =  1153.200  mm,
	W =     5.544 deg,	P =    60.170 deg,	R =  -166.026 deg
   GP2:
	UF : 1, UT : 1,
	J1=    90.000 deg,	J2=    90.000 deg
};
P[382]{
   GP1:
	UF : 1, UT : 1,		CONFIG : 'N U T, 0, 0, 0',
	X =  1686.139  mm,	Y =   462.621  mm,	Z =   834.516  mm,
	W =    39.867 deg,	P =   -22.888 deg,	R =   -65.014 deg
   GP2:
	UF : 1, UT : 1,
	J1=   -90.000 deg,	J2=   -90.000 deg
};
P[383]{
   GP1:
	UF : 1, UT : 1,		CONFIG : 'N U T, 0, 0, 0',
	X =  1686.139  mm,	Y =   476.121  mm,	Z =   834.516  mm,
	W =    39.867 deg,	P =   -22.888 deg,	R =   -65.014 deg
   GP2:
	UF : 1, UT : 1,
	J1=   -90.000 deg,	J2=   -90.000 deg
};
P[384]{
   GP1:
	UF : 1, UT : 1,		CONFIG : 'N U T, 0, 0, 0',
	X =  1685.925  mm,	Y =   479.979  mm,	Z =   834.516  mm,
	W =    39.867 deg,	P =   -22.888 deg,	R =   -69.837 deg
   GP2:
	UF : 1, UT : 1,
	J1=   -90.000 deg,	J2=   -90.000 deg
};
P[385]{
   GP1:
	UF : 1, UT : 1,		CONFIG : 'N U T, 0, 0, 0',
	X =  1687.210  mm,	Y =   484.764  mm,	Z =   834.516  mm,
	W =    39.867 deg,	P =   -22.888 deg,	R =   -70.971 deg
   GP2:
	UF : 1, UT : 1,
	J1=   -90.000 deg,	J2=   -90.000 deg
};
P[386]{
   GP1:
	UF : 1, UT : 1,		CONFIG : 'N U T, 0, 0, 0',
	X =  1712.772  mm,	Y =   557.381  mm,	Z =   832.210  mm,
	W =    39.870 deg,	P =   -22.884 deg,	R =   -70.976 deg
   GP2:
	UF : 1, UT : 1,
	J1=   -90.000 deg,	J2=   -90.000 deg
};
P[387]{
   GP1:
	UF : 1, UT : 1,		CONFIG : 'N U T, 0, 0, 0',
	X =  1714.058  mm,	Y =   562.095  mm,	Z =   832.211  mm,
	W =    39.870 deg,	P =   -22.884 deg,	R =   -74.847 deg
   GP2:
	UF : 1, UT : 1,
	J1=   -90.000 deg,	J2=   -90.000 deg
};
P[388]{
   GP1:
	UF : 1, UT : 1,		CONFIG : 'N U T, 0, 0, 0',
	X =  1597.869  mm,	Y =  -854.871  mm,	Z =   914.402  mm,
	W =   -20.245 deg,	P =   -41.090 deg,	R =    57.299 deg
   GP2:
	UF : 1, UT : 1,
	J1=   -90.000 deg,	J2=    90.000 deg
};
P[389]{
   GP1:
	UF : 1, UT : 1,		CONFIG : 'N U T, 0, 0, 0',
	X =  1597.869  mm,	Y =  -357.729  mm,	Z =   914.402  mm,
	W =   -53.336 deg,	P =     2.108 deg,	R =    49.603 deg
   GP2:
	UF : 1, UT : 1,
	J1=   -90.000 deg,	J2=    90.000 deg
};
P[390]{
   GP1:
	UF : 1, UT : 1,		CONFIG : 'N U T, 0, 0, 0',
	X =  1716.179  mm,	Y =   565.067  mm,	Z =   832.183  mm,
	W =    39.866 deg,	P =   -22.883 deg,	R =   -84.917 deg
   GP2:
	UF : 1, UT : 1,
	J1=   -90.000 deg,	J2=   -90.000 deg
};
P[391]{
   GP1:
	UF : 1, UT : 1,		CONFIG : 'N U T, 0, 0, 0',
	X =  1855.755  mm,	Y =   827.617  mm,	Z =   833.144  mm,
	W =    13.492 deg,	P =   -43.347 deg,	R =   -39.152 deg
   GP2:
	UF : 1, UT : 1,
	J1=   -90.000 deg,	J2=   -90.000 deg
};
P[392]{
   GP1:
	UF : 1, UT : 1,		CONFIG : 'N U T, 0, 0, 0',
	X =  1705.182  mm,	Y =   420.290  mm,	Z =   833.994  mm,
	W =    43.054 deg,	P =   -14.371 deg,	R =   -45.081 deg
   GP2:
	UF : 1, UT : 1,
	J1=   -90.000 deg,	J2=   -90.000 deg
};
P[393]{
   GP1:
	UF : 1, UT : 1,		CONFIG : 'N U T, 0, 0, 0',
	X =  1835.752  mm,	Y =   267.646  mm,	Z =   833.994  mm,
	W =    43.054 deg,	P =   -14.371 deg,	R =   -45.081 deg
   GP2:
	UF : 1, UT : 1,
	J1=   -90.000 deg,	J2=   -90.000 deg
};
P[394]{
   GP1:
	UF : 1, UT : 1,		CONFIG : 'N U T, 0, 0, 0',
	X =  1841.258  mm,	Y =   261.450  mm,	Z =   833.984  mm,
	W =    43.049 deg,	P =   -14.375 deg,	R =   -42.871 deg
   GP2:
	UF : 1, UT : 1,
	J1=   -90.000 deg,	J2=   -90.000 deg
};
P[395]{
   GP1:
	UF : 1, UT : 1,		CONFIG : 'N U T, 0, 0, 0',
	X =  1813.190  mm,	Y =  -222.628  mm,	Z =   892.611  mm,
	W =   -54.261 deg,	P =    -6.374 deg,	R =    77.692 deg
   GP2:
	UF : 1, UT : 1,
	J1=   -90.000 deg,	J2=    90.000 deg
};
P[396]{
   GP1:
	UF : 1, UT : 1,		CONFIG : 'N U T, 0, 0, 0',
	X =  1480.982  mm,	Y =  -280.121  mm,	Z =   888.392  mm,
	W =   -52.435 deg,	P =    -5.968 deg,	R =    77.563 deg
   GP2:
	UF : 1, UT : 1,
	J1=   -90.000 deg,	J2=    90.000 deg
};
P[397]{
   GP1:
	UF : 1, UT : 1,		CONFIG : 'N U T, 0, 0, -1',
	X =  2103.205  mm,	Y =   181.792  mm,	Z =  1015.411  mm,
	W =     -.647 deg,	P =    55.219 deg,	R =   156.602 deg
   GP2:
	UF : 1, UT : 1,
	J1=    90.000 deg,	J2=    90.000 deg
};
P[398]{
   GP1:
	UF : 1, UT : 1,		CONFIG : 'N U T, 0, 0, -1',
	X =  2131.893  mm,	Y =   160.632  mm,	Z =   829.995  mm,
	W =     2.033 deg,	P =    39.456 deg,	R =   159.535 deg
   GP2:
	UF : 1, UT : 1,
	J1=    90.000 deg,	J2=    90.000 deg
};
P[399]{
   GP1:
	UF : 1, UT : 1,		CONFIG : 'N U T, 0, 0, -1',
	X =  2138.420  mm,	Y =   177.761  mm,	Z =   828.017  mm,
	W =     3.162 deg,	P =    39.786 deg,	R =   160.410 deg
   GP2:
	UF : 1, UT : 1,
	J1=    90.000 deg,	J2=    90.000 deg
};
P[400]{
   GP1:
	UF : 1, UT : 1,		CONFIG : 'N U T, 0, 0, 0',
	X =  1854.256  mm,	Y =   251.093  mm,	Z =   833.983  mm,
	W =    43.049 deg,	P =   -14.375 deg,	R =   -40.829 deg
   GP2:
	UF : 1, UT : 1,
	J1=   -90.000 deg,	J2=   -90.000 deg
};
P[401]{
   GP1:
	UF : 1, UT : 1,		CONFIG : 'N U T, 0, 0, 0',
	X =  1914.826  mm,	Y =   204.450  mm,	Z =   834.412  mm,
	W =    43.049 deg,	P =   -14.375 deg,	R =   -40.829 deg
   GP2:
	UF : 1, UT : 1,
	J1=   -90.000 deg,	J2=   -90.000 deg
};
P[402]{
   GP1:
	UF : 1, UT : 1,		CONFIG : 'N U T, 0, 0, 0',
	X =  2126.251  mm,	Y =   205.487  mm,	Z =   828.238  mm,
	W =     2.943 deg,	P =    38.020 deg,	R =  -104.065 deg
   GP2:
	UF : 1, UT : 1,
	J1=    90.000 deg,	J2=    90.000 deg
};
P[403]{
   GP1:
	UF : 1, UT : 1,		CONFIG : 'N U T, 0, 0, 0',
	X =  2099.621  mm,	Y =   193.357  mm,	Z =   825.885  mm,
	W =     -.694 deg,	P =    38.678 deg,	R =   -19.390 deg
   GP2:
	UF : 1, UT : 1,
	J1=    90.000 deg,	J2=    90.000 deg
};
P[404]{
   GP1:
	UF : 1, UT : 1,		CONFIG : 'N U T, 0, 0, 0',
	X =  1687.918  mm,	Y =  -462.979  mm,	Z =   838.919  mm,
	W =   -28.321 deg,	P =   -37.471 deg,	R =    36.648 deg
   GP2:
	UF : 1, UT : 1,
	J1=   -90.000 deg,	J2=    90.000 deg
};
P[405]{
   GP1:
	UF : 1, UT : 1,		CONFIG : 'N U T, 0, 0, 0',
	X =  1688.170  mm,	Y =  -479.676  mm,	Z =   839.279  mm,
	W =   -28.322 deg,	P =   -37.469 deg,	R =    36.650 deg
   GP2:
	UF : 1, UT : 1,
	J1=   -90.000 deg,	J2=    90.000 deg
};
P[406]{
   GP1:
	UF : 1, UT : 1,		CONFIG : 'N U T, 0, 0, 0',
	X =  2086.999  mm,	Y =   153.311  mm,	Z =   827.577  mm,
	W =     -.631 deg,	P =    41.060 deg,	R =   -19.279 deg
   GP2:
	UF : 1, UT : 1,
	J1=    90.000 deg,	J2=    90.000 deg
};
P[407]{
   GP1:
	UF : 1, UT : 1,		CONFIG : 'N U T, 0, 0, 0',
	X =  2099.893  mm,	Y =   128.272  mm,	Z =   828.182  mm,
	W =     2.900 deg,	P =    42.082 deg,	R =    77.981 deg
   GP2:
	UF : 1, UT : 1,
	J1=    90.000 deg,	J2=    90.000 deg
};
P[408]{
   GP1:
	UF : 1, UT : 1,		CONFIG : 'N U T, 0, 0, 0',
	X =  1689.098  mm,	Y =  -484.247  mm,	Z =   837.566  mm,
	W =   -28.322 deg,	P =   -37.469 deg,	R =    39.720 deg
   GP2:
	UF : 1, UT : 1,
	J1=   -90.000 deg,	J2=    90.000 deg
};
P[409]{
   GP1:
	UF : 1, UT : 1,		CONFIG : 'N U T, 0, 0, 0',
	X =  1689.669  mm,	Y =  -488.318  mm,	Z =   837.566  mm,
	W =   -28.322 deg,	P =   -37.469 deg,	R =    41.171 deg
   GP2:
	UF : 1, UT : 1,
	J1=   -90.000 deg,	J2=    90.000 deg
};
P[410]{
   GP1:
	UF : 1, UT : 1,		CONFIG : 'N U T, 0, 0, 0',
	X =  2126.676  mm,	Y =   140.641  mm,	Z =   828.927  mm,
	W =     2.158 deg,	P =    43.251 deg,	R =   161.040 deg
   GP2:
	UF : 1, UT : 1,
	J1=    90.000 deg,	J2=    90.000 deg
};
P[411]{
   GP1:
	UF : 1, UT : 1,		CONFIG : 'N U T, 0, 0, 0',
	X =  2132.026  mm,	Y =   160.981  mm,	Z =   829.412  mm,
	W =     3.206 deg,	P =    40.722 deg,	R =   159.881 deg
   GP2:
	UF : 1, UT : 1,
	J1=    90.000 deg,	J2=    90.000 deg
};
P[412]{
   GP1:
	UF : 1, UT : 1,		CONFIG : 'N U T, 0, 0, 0',
	X =  2054.302  mm,	Y =   204.441  mm,	Z =   988.994  mm,
	W =      .815 deg,	P =    36.667 deg,	R =   159.784 deg
   GP2:
	UF : 1, UT : 1,
	J1=    90.000 deg,	J2=    90.000 deg
};
P[413]{
   GP1:
	UF : 1, UT : 1,		CONFIG : 'N U T, 0, 0, 0',
	X =  2128.801  mm,	Y =   250.942  mm,	Z =   983.493  mm,
	W =    -8.588 deg,	P =    43.492 deg,	R =    86.611 deg
   GP2:
	UF : 1, UT : 1,
	J1=    90.000 deg,	J2=    90.000 deg
};
P[414]{
   GP1:
	UF : 1, UT : 1,		CONFIG : 'N U T, 0, 0, 0',
	X =  2109.036  mm,	Y =   233.060  mm,	Z =   825.919  mm,
	W =    -2.535 deg,	P =    44.944 deg,	R =    86.414 deg
   GP2:
	UF : 1, UT : 1,
	J1=    90.000 deg,	J2=    90.000 deg
};
P[415]{
   GP1:
	UF : 1, UT : 1,		CONFIG : 'N U T, 0, 0, 0',
	X =  1711.454  mm,	Y =  -560.605  mm,	Z =   837.994  mm,
	W =   -28.322 deg,	P =   -37.469 deg,	R =    41.171 deg
   GP2:
	UF : 1, UT : 1,
	J1=   -90.000 deg,	J2=    90.000 deg
};
P[416]{
   GP1:
	UF : 1, UT : 1,		CONFIG : 'N U T, 0, 0, 0',
	X =  1713.167  mm,	Y =  -564.177  mm,	Z =   838.637  mm,
	W =   -28.322 deg,	P =   -37.469 deg,	R =    44.951 deg
   GP2:
	UF : 1, UT : 1,
	J1=   -90.000 deg,	J2=    90.000 deg
};
P[417]{
   GP1:
	UF : 1, UT : 1,		CONFIG : 'N U T, 0, 0, 0',
	X =  1715.596  mm,	Y =  -568.035  mm,	Z =   837.566  mm,
	W =   -28.322 deg,	P =   -37.469 deg,	R =    50.636 deg
   GP2:
	UF : 1, UT : 1,
	J1=   -90.000 deg,	J2=    90.000 deg
};
P[418]{
   GP1:
	UF : 1, UT : 1,		CONFIG : 'N U T, 0, 0, 0',
	X =  2201.411  mm,	Y =   234.520  mm,	Z =   827.585  mm,
	W =    -2.535 deg,	P =    44.944 deg,	R =    86.414 deg
   GP2:
	UF : 1, UT : 1,
	J1=    90.000 deg,	J2=    90.000 deg
};
P[419]{
   GP1:
	UF : 1, UT : 1,		CONFIG : 'N U T, 0, 0, 0',
	X =  2212.981  mm,	Y =   231.980  mm,	Z =   827.741  mm,
	W =    -2.535 deg,	P =    44.943 deg,	R =    56.627 deg
   GP2:
	UF : 1, UT : 1,
	J1=    90.000 deg,	J2=    90.000 deg
};
P[420]{
   GP1:
	UF : 1, UT : 1,		CONFIG : 'N U T, 0, 0, 0',
	X =  1850.878  mm,	Y =  -825.178  mm,	Z =   836.854  mm,
	W =   -28.322 deg,	P =   -37.469 deg,	R =    50.636 deg
   GP2:
	UF : 1, UT : 1,
	J1=   -90.000 deg,	J2=    90.000 deg
};
P[421]{
   GP1:
	UF : 1, UT : 1,		CONFIG : 'N U T, 0, 0, 0',
	X =  1703.240  mm,	Y =  -424.313  mm,	Z =   832.247  mm,
	W =   -39.460 deg,	P =    -8.334 deg,	R =    42.657 deg
   GP2:
	UF : 1, UT : 1,
	J1=   -90.000 deg,	J2=    90.000 deg
};
P[422]{
   GP1:
	UF : 1, UT : 1,		CONFIG : 'N U T, 0, 0, 0',
	X =  1836.384  mm,	Y =  -271.171  mm,	Z =   832.247  mm,
	W =   -39.460 deg,	P =    -8.334 deg,	R =    42.657 deg
   GP2:
	UF : 1, UT : 1,
	J1=   -90.000 deg,	J2=    90.000 deg
};
P[423]{
   GP1:
	UF : 1, UT : 1,		CONFIG : 'N U T, 0, 0, 0',
	X =  2221.646  mm,	Y =   223.084  mm,	Z =   826.750  mm,
	W =     -.368 deg,	P =    44.999 deg,	R =    40.109 deg
   GP2:
	UF : 1, UT : 1,
	J1=    90.000 deg,	J2=    90.000 deg
};
P[424]{
   GP1:
	UF : 1, UT : 1,		CONFIG : 'N U T, 0, 0, 0',
	X =  2447.358  mm,	Y =   -34.111  mm,	Z =   825.303  mm,
	W =     -.103 deg,	P =    45.000 deg,	R =    45.359 deg
   GP2:
	UF : 1, UT : 1,
	J1=    90.000 deg,	J2=    90.000 deg
};
P[425]{
   GP1:
	UF : 1, UT : 1,		CONFIG : 'N U T, 0, 0, 0',
	X =  2449.920  mm,	Y =   -38.165  mm,	Z =   824.850  mm,
	W =     -.103 deg,	P =    45.000 deg,	R =    54.166 deg
   GP2:
	UF : 1, UT : 1,
	J1=    90.000 deg,	J2=    90.000 deg
};
P[426]{
   GP1:
	UF : 1, UT : 1,		CONFIG : 'N U T, 0, 0, 0',
	X =  2457.259  mm,	Y =   -44.429  mm,	Z =   824.725  mm,
	W =     -.103 deg,	P =    45.001 deg,	R =    54.620 deg
   GP2:
	UF : 1, UT : 1,
	J1=    90.000 deg,	J2=    90.000 deg
};
P[427]{
   GP1:
	UF : 1, UT : 1,		CONFIG : 'N U T, 0, 0, 0',
	X =  1843.099  mm,	Y =  -264.599  mm,	Z =   832.247  mm,
	W =   -39.460 deg,	P =    -8.334 deg,	R =    38.620 deg
   GP2:
	UF : 1, UT : 1,
	J1=   -90.000 deg,	J2=    90.000 deg
};
P[428]{
   GP1:
	UF : 1, UT : 1,		CONFIG : 'N U T, 0, 0, 0',
	X =  1858.669  mm,	Y =  -251.384  mm,	Z =   832.248  mm,
	W =   -39.460 deg,	P =    -8.334 deg,	R =    38.620 deg
   GP2:
	UF : 1, UT : 1,
	J1=   -90.000 deg,	J2=    90.000 deg
};
P[429]{
   GP1:
	UF : 1, UT : 1,		CONFIG : 'N U T, 0, 0, 0',
	X =  1912.811  mm,	Y =  -209.527  mm,	Z =   832.247  mm,
	W =   -39.460 deg,	P =    -8.334 deg,	R =    45.243 deg
   GP2:
	UF : 1, UT : 1,
	J1=   -90.000 deg,	J2=    90.000 deg
};
P[430]{
   GP1:
	UF : 1, UT : 1,		CONFIG : 'N U T, 0, 0, 0',
	X =  2645.400  mm,	Y =  -183.513  mm,	Z =   824.417  mm,
	W =   -30.972 deg,	P =    27.486 deg,	R =    12.662 deg
   GP2:
	UF : 1, UT : 1,
	J1=    90.000 deg,	J2=    90.000 deg
};
P[431]{
   GP1:
	UF : 1, UT : 1,		CONFIG : 'N U T, 0, 0, 0',
	X =  2669.763  mm,	Y =  -202.477  mm,	Z =   824.028  mm,
	W =   -30.972 deg,	P =    27.486 deg,	R =    12.662 deg
   GP2:
	UF : 1, UT : 1,
	J1=    90.000 deg,	J2=    90.000 deg
};
P[432]{
   GP1:
	UF : 1, UT : 1,		CONFIG : 'N U T, 0, 0, 0',
	X =  2643.424  mm,	Y =  -135.910  mm,	Z =   990.550  mm,
	W =   -36.400 deg,	P =    28.534 deg,	R =    31.709 deg
   GP2:
	UF : 1, UT : 1,
	J1=    90.000 deg,	J2=    90.000 deg
};
P[433]{
   GP1:
	UF : 1, UT : 1,		CONFIG : 'N U T, 0, 0, 0',
	X =   983.140  mm,	Y =    19.420  mm,	Z =   990.550  mm,
	W =   -36.400 deg,	P =    28.534 deg,	R =    23.998 deg
   GP2:
	UF : 1, UT : 1,
	J1=    90.000 deg,	J2=    90.000 deg
};
P[434]{
   GP1:
	UF : 1, UT : 1,		CONFIG : 'N U T, 0, 0, 0',
	X =   983.140  mm,	Y =  -212.416  mm,	Z =   990.550  mm,
	W =   -43.636 deg,	P =   -12.296 deg,	R =    70.660 deg
   GP2:
	UF : 1, UT : 1,
	J1=    80.000 deg,	J2=    90.000 deg
};
P[435]{
   GP1:
	UF : 1, UT : 1,		CONFIG : 'N U T, 0, 0, 0',
	X =  1995.140  mm,	Y =  -212.416  mm,	Z =   320.550  mm,
	W =   -43.636 deg,	P =   -12.296 deg,	R =    70.660 deg
   GP2:
	UF : 1, UT : 1,
	J1=    80.000 deg,	J2=    90.000 deg
};
P[436]{
   GP1:
	UF : 1, UT : 1,		CONFIG : 'N U T, 0, 0, 0',
	X =  2018.730  mm,	Y =   -25.769  mm,	Z =   130.343  mm,
	W =   -38.665 deg,	P =    -2.420 deg,	R =   142.728 deg
   GP2:
	UF : 1, UT : 1,
	J1=    80.000 deg,	J2=    90.000 deg
};
P[437]{
   GP1:
	UF : 1, UT : 1,		CONFIG : 'N U T, 0, 0, 0',
	X =  2072.355  mm,	Y =    35.409  mm,	Z =    15.812  mm,
	W =   -31.287 deg,	P =    -2.153 deg,	R =   142.523 deg
   GP2:
	UF : 1, UT : 1,
	J1=    80.000 deg,	J2=    90.000 deg
};
P[438]{
   GP1:
	UF : 1, UT : 1,		CONFIG : 'N U T, 0, 0, 0',
	X =  2107.225  mm,	Y =     1.061  mm,	Z =     8.326  mm,
	W =   -27.569 deg,	P =     5.116 deg,	R =   142.904 deg
   GP2:
	UF : 1, UT : 1,
	J1=    80.000 deg,	J2=    90.000 deg
};
P[439]{
   GP1:
	UF : 1, UT : 1,		CONFIG : 'N U T, 0, 0, 0',
	X =  2110.724  mm,	Y =    -1.284  mm,	Z =     7.786  mm,
	W =   -27.578 deg,	P =     5.122 deg,	R =   139.594 deg
   GP2:
	UF : 1, UT : 1,
	J1=    80.000 deg,	J2=    90.000 deg
};
P[440]{
   GP1:
	UF : 1, UT : 1,		CONFIG : 'N U T, 0, 0, 0',
	X =  2115.361  mm,	Y =    -5.660  mm,	Z =     5.643  mm,
	W =   -27.580 deg,	P =     5.121 deg,	R =   136.987 deg
   GP2:
	UF : 1, UT : 1,
	J1=    80.000 deg,	J2=    90.000 deg
};
P[441]{
   GP1:
	UF : 1, UT : 1,		CONFIG : 'N U T, 0, 0, 0',
	X =  2245.407  mm,	Y =  -182.117  mm,	Z =   -16.249  mm,
	W =   -36.469 deg,	P =    -8.806 deg,	R =   122.593 deg
   GP2:
	UF : 1, UT : 1,
	J1=    80.000 deg,	J2=    90.000 deg
};
P[442]{
   GP1:
	UF : 1, UT : 1,		CONFIG : 'N U T, 0, 0, 0',
	X =  2249.594  mm,	Y =  -187.703  mm,	Z =   -16.744  mm,
	W =   -36.562 deg,	P =   -11.678 deg,	R =   125.987 deg
   GP2:
	UF : 1, UT : 1,
	J1=    80.000 deg,	J2=    90.000 deg
};
P[443]{
   GP1:
	UF : 1, UT : 1,		CONFIG : 'N U T, 0, 0, 0',
	X =  2258.662  mm,	Y =  -198.230  mm,	Z =   -16.565  mm,
	W =   -36.304 deg,	P =   -14.505 deg,	R =   128.304 deg
   GP2:
	UF : 1, UT : 1,
	J1=    80.000 deg,	J2=    90.000 deg
};
P[444]{
   GP1:
	UF : 1, UT : 1,		CONFIG : 'N U T, 0, 0, 0',
	X =  2506.162  mm,	Y =  -435.146  mm,	Z =   -55.106  mm,
	W =   -23.402 deg,	P =   -31.777 deg,	R =    95.143 deg
   GP2:
	UF : 1, UT : 1,
	J1=    80.000 deg,	J2=    90.000 deg
};
P[445]{
   GP1:
	UF : 1, UT : 1,		CONFIG : 'N U T, 0, 0, 0',
	X =  2519.709  mm,	Y =  -443.017  mm,	Z =   -58.897  mm,
	W =   -18.439 deg,	P =   -37.731 deg,	R =   100.757 deg
   GP2:
	UF : 1, UT : 1,
	J1=    80.000 deg,	J2=    90.000 deg
};
P[446]{
   GP1:
	UF : 1, UT : 1,		CONFIG : 'N U T, 0, 0, 0',
	X =  2541.609  mm,	Y =  -449.213  mm,	Z =   -62.962  mm,
	W =   -18.799 deg,	P =   -40.099 deg,	R =   104.558 deg
   GP2:
	UF : 1, UT : 1,
	J1=    80.000 deg,	J2=    90.000 deg
};
P[447]{
   GP1:
	UF : 1, UT : 1,		CONFIG : 'N U T, 0, 0, 0',
	X =  2557.851  mm,	Y =  -453.975  mm,	Z =   -64.097  mm,
	W =   -18.770 deg,	P =   -39.987 deg,	R =   104.546 deg
   GP2:
	UF : 1, UT : 1,
	J1=    80.000 deg,	J2=    90.000 deg
};
P[448]{
   GP1:
	UF : 1, UT : 1,		CONFIG : 'N U T, 0, 0, 0',
	X =  2603.552  mm,	Y =  -487.198  mm,	Z =   -75.346  mm,
	W =   -35.254 deg,	P =   -23.937 deg,	R =   103.286 deg
   GP2:
	UF : 1, UT : 1,
	J1=    80.000 deg,	J2=    90.000 deg
};
P[449]{
   GP1:
	UF : 1, UT : 1,		CONFIG : 'N U T, 0, 0, 0',
	X =  2619.220  mm,	Y =  -522.655  mm,	Z =   -84.357  mm,
	W =   -33.010 deg,	P =   -16.169 deg,	R =    63.148 deg
   GP2:
	UF : 1, UT : 1,
	J1=    80.000 deg,	J2=    90.000 deg
};
P[450]{
   GP1:
	UF : 1, UT : 1,		CONFIG : 'N U T, 0, 0, 0',
	X =  2618.055  mm,	Y =  -722.080  mm,	Z =   -81.773  mm,
	W =   -27.680 deg,	P =   -22.323 deg,	R =    54.101 deg
   GP2:
	UF : 1, UT : 1,
	J1=    80.000 deg,	J2=    90.000 deg
};
P[451]{
   GP1:
	UF : 1, UT : 1,		CONFIG : 'N U T, 0, 0, 0',
	X =  2562.114  mm,	Y =  -708.403  mm,	Z =     7.893  mm,
	W =   -27.687 deg,	P =   -22.321 deg,	R =    54.103 deg
   GP2:
	UF : 1, UT : 1,
	J1=    80.000 deg,	J2=    90.000 deg
};
P[452]{
   GP1:
	UF : 1, UT : 1,		CONFIG : 'N U T, 0, 0, 0',
	X =  2517.838  mm,	Y =  -811.403  mm,	Z =     7.893  mm,
	W =   -27.687 deg,	P =   -22.321 deg,	R =    54.103 deg
   GP2:
	UF : 1, UT : 1,
	J1=    80.000 deg,	J2=    90.000 deg
};
P[453]{
   GP1:
	UF : 1, UT : 1,		CONFIG : 'N U T, 0, 0, 0',
	X =  2546.452  mm,	Y =  -827.140  mm,	Z =   -68.564  mm,
	W =   -27.686 deg,	P =   -22.321 deg,	R =    54.103 deg
   GP2:
	UF : 1, UT : 1,
	J1=    80.000 deg,	J2=    90.000 deg
};
P[454]{
   GP1:
	UF : 1, UT : 1,		CONFIG : 'N U T, 0, 0, 0',
	X =  2547.367  mm,	Y =  -816.426  mm,	Z =   -70.480  mm,
	W =   -27.686 deg,	P =   -22.321 deg,	R =    54.103 deg
   GP2:
	UF : 1, UT : 1,
	J1=    80.000 deg,	J2=    90.000 deg
};
P[455]{
   GP1:
	UF : 1, UT : 1,		CONFIG : 'N U T, 0, 0, 0',
	X =  2551.667  mm,	Y =  -807.998  mm,	Z =   -72.144  mm,
	W =   -35.030 deg,	P =    -5.089 deg,	R =    46.504 deg
   GP2:
	UF : 1, UT : 1,
	J1=    80.000 deg,	J2=    90.000 deg
};
P[456]{
   GP1:
	UF : 1, UT : 1,		CONFIG : 'N U T, 0, 0, 0',
	X =  2563.152  mm,	Y =  -800.022  mm,	Z =   -73.315  mm,
	W =   -35.920 deg,	P =     6.424 deg,	R =    38.938 deg
   GP2:
	UF : 1, UT : 1,
	J1=    80.000 deg,	J2=    90.000 deg
};
P[457]{
   GP1:
	UF : 1, UT : 1,		CONFIG : 'N U T, 0, 0, 0',
	X =  2604.094  mm,	Y =  -768.658  mm,	Z =   -79.200  mm,
	W =   -30.378 deg,	P =    -1.294 deg,	R =    48.839 deg
   GP2:
	UF : 1, UT : 1,
	J1=    80.000 deg,	J2=    90.000 deg
};
P[458]{
   GP1:
	UF : 1, UT : 1,		CONFIG : 'N U T, 0, 0, 0',
	X =  2620.852  mm,	Y =  -723.431  mm,	Z =   -82.347  mm,
	W =   -25.591 deg,	P =   -24.735 deg,	R =    48.858 deg
   GP2:
	UF : 1, UT : 1,
	J1=    80.000 deg,	J2=    90.000 deg
};
P[459]{
   GP1:
	UF : 1, UT : 1,		CONFIG : 'N U T, 0, 0, 0',
	X =  2551.662  mm,	Y =  -712.821  mm,	Z =   124.119  mm,
	W =   -35.203 deg,	P =   -31.584 deg,	R =    53.410 deg
   GP2:
	UF : 1, UT : 1,
	J1=    80.000 deg,	J2=    90.000 deg
};
P[460]{
   GP1:
	UF : 1, UT : 1,		CONFIG : 'N U T, 0, 0, 0',
	X =  1870.645  mm,	Y =  -712.821  mm,	Z =   348.203  mm,
	W =   -35.203 deg,	P =   -31.584 deg,	R =    53.410 deg
   GP2:
	UF : 1, UT : 1,
	J1=    80.000 deg,	J2=    90.000 deg
};
P[461]{
   GP1:
	UF : 1, UT : 1,		CONFIG : 'N U T, 0, 0, 0',
	X =   472.370  mm,	Y = -1534.903  mm,	Z =   492.380  mm,
	W =    50.539 deg,	P =     3.993 deg,	R =   -65.902 deg
   GP2:
	UF : 1, UT : 1,
	J1=    80.000 deg,	J2=    90.000 deg
};
P[462]{
   GP1:
	UF : 1, UT : 1,		CONFIG : 'N U T, 0, 0, 0',
	X =  2789.986  mm,	Y = -1514.458  mm,	Z =   933.459  mm,
	W =   -37.771 deg,	P =   -31.405 deg,	R =    42.828 deg
   GP2:
	UF : 1, UT : 1,
	J1=   100.000 deg,	J2=   -90.000 deg
};
P[463]{
   GP1:
	UF : 1, UT : 1,		CONFIG : 'N U T, 0, 0, 0',
	X =  2785.008  mm,	Y = -1534.382  mm,	Z =   930.705  mm,
	W =   -42.870 deg,	P =   -22.985 deg,	R =    43.312 deg
   GP2:
	UF : 1, UT : 1,
	J1=   100.000 deg,	J2=   -90.000 deg
};
P[464]{
   GP1:
	UF : 1, UT : 1,		CONFIG : 'N U T, 0, 0, 0',
	X =  2768.811  mm,	Y = -1552.001  mm,	Z =   928.547  mm,
	W =   -45.718 deg,	P =   -14.892 deg,	R =    35.274 deg
   GP2:
	UF : 1, UT : 1,
	J1=   100.000 deg,	J2=   -90.000 deg
};
P[465]{
   GP1:
	UF : 1, UT : 1,		CONFIG : 'N U T, 0, 0, 0',
	X =  2729.736  mm,	Y = -1572.169  mm,	Z =   921.941  mm,
	W =   -45.718 deg,	P =   -14.891 deg,	R =    30.406 deg
   GP2:
	UF : 1, UT : 1,
	J1=   100.000 deg,	J2=   -90.000 deg
};
P[466]{
   GP1:
	UF : 1, UT : 1,		CONFIG : 'N U T, 0, 0, 0',
	X =  2716.465  mm,	Y = -1576.342  mm,	Z =   919.062  mm,
	W =   -45.718 deg,	P =   -14.891 deg,	R =    18.309 deg
   GP2:
	UF : 1, UT : 1,
	J1=   100.000 deg,	J2=   -90.000 deg
};
P[467]{
   GP1:
	UF : 1, UT : 1,		CONFIG : 'N U T, 0, 0, 0',
	X =  2710.176  mm,	Y = -1578.011  mm,	Z =   916.890  mm,
	W =   -45.718 deg,	P =   -14.891 deg,	R =     6.077 deg
   GP2:
	UF : 1, UT : 1,
	J1=   100.000 deg,	J2=   -90.000 deg
};
P[468]{
   GP1:
	UF : 1, UT : 1,		CONFIG : 'N U T, 0, 0, 0',
	X =  2679.569  mm,	Y = -1578.685  mm,	Z =   910.803  mm,
	W =   -43.507 deg,	P =   -15.108 deg,	R =     5.505 deg
   GP2:
	UF : 1, UT : 1,
	J1=   100.000 deg,	J2=   -90.000 deg
};
P[469]{
   GP1:
	UF : 1, UT : 1,		CONFIG : 'N U T, 0, 0, 0',
	X =  2612.111  mm,	Y = -1537.301  mm,	Z =  1175.202  mm,
	W =   -45.531 deg,	P =     6.252 deg,	R =    32.963 deg
   GP2:
	UF : 0, UT : 1,
	J1=   100.000 deg,	J2=   -90.000 deg
};
P[470]{
   GP1:
	UF : 1, UT : 1,		CONFIG : 'N U T, 0, 0, 0',
	X =  2071.007  mm,	Y = -1554.081  mm,	Z =  1677.384  mm,
	W =   -46.027 deg,	P =   -17.509 deg,	R =    23.991 deg
   GP2:
	UF : 1, UT : 1,
	J1=   100.000 deg,	J2=   -90.000 deg
};
P[471]{
   GP1:
	UF : 1, UT : 1,		CONFIG : 'N U T, 0, 0, 0',
	X =  1642.115  mm,	Y = -1225.593  mm,	Z =  1744.283  mm,
	W =   -30.785 deg,	P =   -19.925 deg,	R =    38.701 deg
   GP2:
	UF : 1, UT : 1,
	J1=   100.000 deg,	J2=   -90.000 deg
};
P[472]{
   GP1:
	UF : 1, UT : 1,		CONFIG : 'N U T, 0, 0, 0',
	X =  1044.179  mm,	Y =  -508.261  mm,	Z =   989.448  mm,
	W =    -7.948 deg,	P =   -16.175 deg,	R =    52.319 deg
   GP2:
	UF : 1, UT : 1,
	J1=   100.000 deg,	J2=   -90.000 deg
};
P[473]{
   GP1:
	UF : 1, UT : 1,		CONFIG : 'N U T, 0, 0, 0',
	X =  2659.725  mm,	Y =  1505.803  mm,	Z =  1079.609  mm,
	W =    15.908 deg,	P =   -31.536 deg,	R =   -26.500 deg
   GP2:
	UF : 0, UT : 1,
	J1=    95.000 deg,	J2=    90.000 deg
};
P[474]{
   GP1:
	UF : 1, UT : 1,		CONFIG : 'N U T, 0, 0, 0',
	X =  2835.237  mm,	Y =  1482.005  mm,	Z =   876.521  mm,
	W =     1.862 deg,	P =   -42.072 deg,	R =    -2.894 deg
   GP2:
	UF : 1, UT : 1,
	J1=    95.000 deg,	J2=    90.000 deg
};
P[475]{
   GP1:
	UF : 1, UT : 1,		CONFIG : 'N U T, 0, 0, 0',
	X =  2835.140  mm,	Y =  1509.059  mm,	Z =   876.904  mm,
	W =      .428 deg,	P =   -42.104 deg,	R =     -.755 deg
   GP2:
	UF : 1, UT : 1,
	J1=    95.000 deg,	J2=    90.000 deg
};
P[476]{
   GP1:
	UF : 1, UT : 1,		CONFIG : 'N U T, 0, 0, 0',
	X =  2829.219  mm,	Y =  1536.845  mm,	Z =   871.630  mm,
	W =    47.771 deg,	P =   -12.839 deg,	R =   -44.177 deg
   GP2:
	UF : 1, UT : 1,
	J1=    95.000 deg,	J2=    90.000 deg
};
P[477]{
   GP1:
	UF : 1, UT : 1,		CONFIG : 'N U T, 0, 0, -1',
	X =  1225.021  mm,	Y = -1373.581  mm,	Z =   228.769  mm,
	W =   -54.518 deg,	P =     8.477 deg,	R =    24.180 deg
   GP2:
	UF : 1, UT : 1,
	J1=    90.000 deg,	J2=   -90.000 deg
};
P[478]{
   GP1:
	UF : 1, UT : 1,		CONFIG : 'N U T, 0, 0, -1',
	X =  2082.302  mm,	Y = -1064.969  mm,	Z =   253.594  mm,
	W =   -44.935 deg,	P =    -7.056 deg,	R =    83.172 deg
   GP2:
	UF : 1, UT : 1,
	J1=    90.000 deg,	J2=   -90.000 deg
};
P[479]{
   GP1:
	UF : 1, UT : 1,		CONFIG : 'N U T, 0, 0, -1',
	X =  2341.243  mm,	Y =  -989.972  mm,	Z =   103.893  mm,
	W =   -44.578 deg,	P =    -6.914 deg,	R =    83.049 deg
   GP2:
	UF : 1, UT : 1,
	J1=    90.000 deg,	J2=   -90.000 deg
};
P[480]{
   GP1:
	UF : 1, UT : 1,		CONFIG : 'N U T, 0, 0, -1',
	X =  2449.739  mm,	Y =  -869.683  mm,	Z =    46.520  mm,
	W =   -44.665 deg,	P =    -6.870 deg,	R =    84.747 deg
   GP2:
	UF : 1, UT : 1,
	J1=    90.000 deg,	J2=   -90.000 deg
};
P[481]{
   GP1:
	UF : 1, UT : 1,		CONFIG : 'N U T, 0, 0, 0',
	X =  2810.648  mm,	Y =  1551.850  mm,	Z =   873.285  mm,
	W =    47.469 deg,	P =    -2.511 deg,	R =   -28.096 deg
   GP2:
	UF : 1, UT : 1,
	J1=    95.000 deg,	J2=    90.000 deg
};
P[482]{
   GP1:
	UF : 1, UT : 1,		CONFIG : 'N U T, 0, 0, 0',
	X =  2772.234  mm,	Y =  1573.304  mm,	Z =   867.965  mm,
	W =    47.469 deg,	P =    -2.511 deg,	R =   -28.096 deg
   GP2:
	UF : 1, UT : 1,
	J1=    95.000 deg,	J2=    90.000 deg
};
P[483]{
   GP1:
	UF : 1, UT : 1,		CONFIG : 'N U T, 0, 0, 0',
	X =  2388.903  mm,	Y =  -813.009  mm,	Z =   289.336  mm,
	W =   -74.527 deg,	P =    19.606 deg,	R =   116.637 deg
   GP2:
	UF : 1, UT : 1,
	J1=    90.000 deg,	J2=   -90.000 deg
};
P[484]{
   GP1:
	UF : 1, UT : 1,		CONFIG : 'N U T, 0, 0, 0',
	X =  2319.444  mm,	Y =  -496.566  mm,	Z =   203.241  mm,
	W =    16.540 deg,	P =   -14.582 deg,	R =      .664 deg
   GP2:
	UF : 1, UT : 1,
	J1=    90.000 deg,	J2=   -90.000 deg
};
P[485]{
   GP1:
	UF : 1, UT : 1,		CONFIG : 'N U T, 0, 0, -1',
	X =  2429.174  mm,	Y =  -689.084  mm,	Z =   108.498  mm,
	W =   -41.825 deg,	P =    18.388 deg,	R =    51.054 deg
   GP2:
	UF : 1, UT : 1,
	J1=    90.000 deg,	J2=   -90.000 deg
};
P[486]{
   GP1:
	UF : 1, UT : 1,		CONFIG : 'N U T, 0, 0, 0',
	X =  2761.802  mm,	Y =  1575.020  mm,	Z =   866.967  mm,
	W =    46.964 deg,	P =     8.280 deg,	R =   -26.942 deg
   GP2:
	UF : 1, UT : 1,
	J1=    95.000 deg,	J2=    90.000 deg
};
P[487]{
   GP1:
	UF : 1, UT : 1,		CONFIG : 'N U T, 0, 0, 0',
	X =  2752.445  mm,	Y =  1575.878  mm,	Z =   865.538  mm,
	W =    46.312 deg,	P =    12.118 deg,	R =   -20.583 deg
   GP2:
	UF : 1, UT : 1,
	J1=    95.000 deg,	J2=    90.000 deg
};
P[488]{
   GP1:
	UF : 1, UT : 1,		CONFIG : 'N U T, 0, 0, 0',
	X =  2431.074  mm,	Y =  -699.084  mm,	Z =   106.298  mm,
	W =   -41.825 deg,	P =    18.388 deg,	R =    51.054 deg
   GP2:
	UF : 1, UT : 1,
	J1=    90.000 deg,	J2=   -90.000 deg
};
P[489]{
   GP1:
	UF : 1, UT : 1,		CONFIG : 'N U T, 0, 0, 0',
	X =  2429.174  mm,	Y =  -689.084  mm,	Z =   254.213  mm,
	W =   -57.120 deg,	P =     5.483 deg,	R =    47.853 deg
   GP2:
	UF : 1, UT : 1,
	J1=    90.000 deg,	J2=   -90.000 deg
};
P[490]{
   GP1:
	UF : 1, UT : 1,		CONFIG : 'N U T, 0, 0, 0',
	X =  1400.602  mm,	Y =  -689.084  mm,	Z =   254.213  mm,
	W =   -57.120 deg,	P =     5.483 deg,	R =    47.853 deg
   GP2:
	UF : 1, UT : 1,
	J1=    90.000 deg,	J2=   -90.000 deg
};
P[491]{
   GP1:
	UF : 1, UT : 1,		CONFIG : 'N U T, 0, 0, 0',
	X =  1400.602  mm,	Y =  -353.084  mm,	Z =   501.233  mm,
	W =    -2.074 deg,	P =   -10.233 deg,	R =    32.173 deg
   GP2:
	UF : 1, UT : 1,
	J1=    90.000 deg,	J2=  -135.000 deg
};
P[492]{
   GP1:
	UF : 1, UT : 1,		CONFIG : 'N U T, 0, 0, 0',
	X =  2655.602  mm,	Y =  -166.084  mm,	Z =   342.233  mm,
	W =     1.417 deg,	P =   -10.343 deg,	R =    12.808 deg
   GP2:
	UF : 1, UT : 1,
	J1=    90.000 deg,	J2=  -135.000 deg
};
P[493]{
   GP1:
	UF : 1, UT : 1,		CONFIG : 'N U T, 0, 0, 0',
	X =  2721.058  mm,	Y =  1576.622  mm,	Z =   862.352  mm,
	W =    46.312 deg,	P =    12.118 deg,	R =   -20.583 deg
   GP2:
	UF : 1, UT : 1,
	J1=    95.000 deg,	J2=    90.000 deg
};
P[494]{
   GP1:
	UF : 1, UT : 1,		CONFIG : 'N U T, 0, 0, 0',
	X =  2586.641  mm,	Y =  1526.023  mm,	Z =  1082.786  mm,
	W =    42.689 deg,	P =    16.599 deg,	R =   -42.374 deg
   GP2:
	UF : 0, UT : 1,
	J1=    95.000 deg,	J2=    90.000 deg
};
P[495]{
   GP1:
	UF : 1, UT : 1,		CONFIG : 'N U T, 0, 0, 0',
	X =  2823.448  mm,	Y =  -159.890  mm,	Z =   258.839  mm,
	W =    -7.346 deg,	P =   -29.104 deg,	R =    14.845 deg
   GP2:
	UF : 1, UT : 1,
	J1=    90.000 deg,	J2=  -135.000 deg
};
P[496]{
   GP1:
	UF : 1, UT : 1,		CONFIG : 'N U T, 0, 0, 0',
	X =  2357.965  mm,	Y =  -270.302  mm,	Z =   258.839  mm,
	W =    -1.017 deg,	P =    -4.421 deg,	R =    12.975 deg
   GP2:
	UF : 1, UT : 1,
	J1=    90.000 deg,	J2=  -135.000 deg
};
P[497]{
   GP1:
	UF : 1, UT : 1,		CONFIG : 'N U T, 0, 0, 0',
	X =  1536.098  mm,	Y =  1365.318  mm,	Z =  1433.705  mm,
	W =    42.689 deg,	P =    16.599 deg,	R =   -30.305 deg
   GP2:
	UF : 1, UT : 1,
	J1=    95.000 deg,	J2=    90.000 deg
};
P[498]{
   GP1:
	UF : 1, UT : 1,		CONFIG : 'N U T, 0, 0, 0',
	X =   498.430  mm,	Y =  -249.509  mm,	Z =  2387.961  mm,
	W =     2.736 deg,	P =   -33.821 deg,	R =   -22.668 deg
   GP2:
	UF : 1, UT : 1,
	J1=    80.000 deg,	J2=    90.000 deg
};
P[499]{
   GP1:
	UF : 1, UT : 1,		CONFIG : 'N U T, 0, 0, 0',
	X =  2641.832  mm,	Y =  -264.435  mm,	Z =   263.645  mm,
	W =     0.000 deg,	P =    -6.880 deg,	R =    -2.940 deg
   GP2:
	UF : 1, UT : 1,
	J1=    90.000 deg,	J2=  -135.000 deg
};
P[500]{
   GP1:
	UF : 1, UT : 1,		CONFIG : 'N U T, 0, 0, 0',
	X =  2474.831  mm,	Y =   -41.435  mm,	Z =    90.241  mm,
	W =    43.945 deg,	P =   -11.174 deg,	R =     1.639 deg
   GP2:
	UF : 1, UT : 1,
	J1=    90.000 deg,	J2=   -90.000 deg
};
P[501]{
   GP1:
	UF : 1, UT : 1,		CONFIG : 'N U T, 0, 0, 0',
	X =  2474.831  mm,	Y =    90.943  mm,	Z =    79.910  mm,
	W =    39.708 deg,	P =   -23.339 deg,	R =    15.773 deg
   GP2:
	UF : 1, UT : 1,
	J1=    90.000 deg,	J2=   -90.000 deg
};
P[502]{
   GP1:
	UF : 1, UT : 1,		CONFIG : 'N U T, 0, 0, 0',
	X =  1773.758  mm,	Y =  1132.590  mm,	Z =   293.935  mm,
	W =   -17.776 deg,	P =    15.458 deg,	R =    47.254 deg
   GP2:
	UF : 1, UT : 1,
	J1=    90.000 deg,	J2=    90.000 deg
};
P[503]{
   GP1:
	UF : 1, UT : 1,		CONFIG : 'N U T, 0, 0, -1',
	X =  1391.376  mm,	Y = -1411.270  mm,	Z =  1335.234  mm,
	W =   -82.179 deg,	P =     1.788 deg,	R =    24.906 deg
   GP2:
	UF : 1, UT : 1,
	J1=    90.000 deg,	J2=   -90.000 deg
};
P[504]{
   GP1:
	UF : 1, UT : 1,		CONFIG : 'N U B, 0, 0, 0',
	X =   357.030  mm,	Y =     -.134  mm,	Z =  2422.493  mm,
	W =     -.020 deg,	P =   -39.773 deg,	R =      .020 deg
   GP2:
	UF : 1, UT : 1,
	J1=    90.000 deg,	J2=    90.000 deg
};
P[505]{
   GP1:
	UF : 1, UT : 1,		CONFIG : 'N U T, 0, 0, 0',
	X =  2478.831  mm,	Y =    82.943  mm,	Z =    74.910  mm,
	W =    39.708 deg,	P =   -23.339 deg,	R =    15.773 deg
   GP2:
	UF : 1, UT : 1,
	J1=    90.000 deg,	J2=   -90.000 deg
};
P[506]{
   GP1:
	UF : 1, UT : 1,		CONFIG : 'N U T, 0, 0, 0',
	X =  2474.831  mm,	Y =  -180.721  mm,	Z =    90.242  mm,
	W =    43.034 deg,	P =    14.904 deg,	R =   -25.132 deg
   GP2:
	UF : 1, UT : 1,
	J1=    90.000 deg,	J2=   -90.000 deg
};
P[507]{
   GP1:
	UF : 1, UT : 1,		CONFIG : 'N U T, 0, 0, 0',
	X =  1656.260  mm,	Y =  -180.721  mm,	Z =    90.242  mm,
	W =    43.034 deg,	P =    14.904 deg,	R =   -25.132 deg
   GP2:
	UF : 1, UT : 1,
	J1=    90.000 deg,	J2=   -90.000 deg
};
P[508]{
   GP1:
	UF : 1, UT : 1,		CONFIG : 'N U B, 0, 0, 0',
	X =   357.030  mm,	Y =     -.134  mm,	Z =  2422.493  mm,
	W =     -.020 deg,	P =   -39.773 deg,	R =      .020 deg
   GP2:
	UF : 1, UT : 1,
	J1=    90.000 deg,	J2=   -90.000 deg
};
P[511]{
   GP1:
	UF : 1, UT : 1,		CONFIG : 'N U T, 0, 0, -1',
	X =  2491.415  mm,	Y =  -851.247  mm,	Z =    -6.408  mm,
	W =   -44.580 deg,	P =    -6.907 deg,	R =    84.735 deg
   GP2:
	UF : 1, UT : 1,
	J1=    90.000 deg,	J2=   -90.000 deg
};
P[512]{
   GP1:
	UF : 1, UT : 1,		CONFIG : 'N U T, 0, 0, -1',
	X =  2491.416  mm,	Y =  -781.247  mm,	Z =    -6.408  mm,
	W =   -44.580 deg,	P =    -6.907 deg,	R =    84.735 deg
   GP2:
	UF : 1, UT : 1,
	J1=    90.000 deg,	J2=   -90.000 deg
};
P[513]{
   GP1:
	UF : 1, UT : 1,		CONFIG : 'N U T, 0, 0, 0',
	X =  2517.662  mm,	Y =  -755.205  mm,	Z =    -9.805  mm,
	W =   -42.771 deg,	P =    15.579 deg,	R =    16.183 deg
   GP2:
	UF : 1, UT : 1,
	J1=    90.000 deg,	J2=   -90.000 deg
};
P[514]{
   GP1:
	UF : 1, UT : 1,		CONFIG : 'N U T, 0, 0, 0',
	X =  2561.304  mm,	Y =  -755.205  mm,	Z =    -9.805  mm,
	W =   -42.771 deg,	P =    15.579 deg,	R =    16.183 deg
   GP2:
	UF : 1, UT : 1,
	J1=    90.000 deg,	J2=   -90.000 deg
};
P[515]{
   GP1:
	UF : 1, UT : 1,		CONFIG : 'N U T, 0, 0, 0',
	X =  2749.284  mm,	Y =  -163.686  mm,	Z =   173.857  mm,
	W =    -1.650 deg,	P =    -7.145 deg,	R =    13.037 deg
   GP2:
	UF : 1, UT : 1,
	J1=    90.000 deg,	J2=  -135.000 deg
};
P[516]{
   GP1:
	UF : 1, UT : 1,		CONFIG : 'N U T, 0, 0, 0',
	X =  2866.388  mm,	Y =  -164.496  mm,	Z =   175.781  mm,
	W =    -5.453 deg,	P =   -22.507 deg,	R =    14.015 deg
   GP2:
	UF : 1, UT : 1,
	J1=    90.000 deg,	J2=  -135.000 deg
};
P[517]{
   GP1:
	UF : 1, UT : 1,		CONFIG : 'N U T, 0, 0, 0',
	X =  2375.248  mm,	Y =  -268.003  mm,	Z =    85.683  mm,
	W =     0.000 deg,	P =     0.000 deg,	R =    -2.940 deg
   GP2:
	UF : 1, UT : 1,
	J1=    90.000 deg,	J2=  -135.000 deg
};
P[518]{
   GP1:
	UF : 1, UT : 1,		CONFIG : 'N U T, 0, 0, 0',
	X =  2746.854  mm,	Y =  -268.663  mm,	Z =    85.683  mm,
	W =     0.000 deg,	P =     0.000 deg,	R =    -2.940 deg
   GP2:
	UF : 1, UT : 1,
	J1=    90.000 deg,	J2=  -135.000 deg
};
P[519]{
   GP1:
	UF : 1, UT : 1,		CONFIG : 'N U T, 0, 0, 0',
	X =  1477.103  mm,	Y =  -165.683  mm,	Z =   137.951  mm,
	W =    38.761 deg,	P =    24.667 deg,	R =   -44.781 deg
   GP2:
	UF : 1, UT : 1,
	J1=    90.000 deg,	J2=   -90.000 deg
};
P[520]{
   GP1:
	UF : 1, UT : 1,		CONFIG : 'N U T, 0, 0, 0',
	X =  2334.769  mm,	Y =  -176.256  mm,	Z =   129.823  mm,
	W =    49.996 deg,	P =    12.253 deg,	R =   -42.841 deg
   GP2:
	UF : 1, UT : 1,
	J1=    90.000 deg,	J2=   -90.000 deg
};
P[521]{
   GP1:
	UF : 1, UT : 1,		CONFIG : 'N U T, 0, 0, 0',
	X =  2334.769  mm,	Y =    95.744  mm,	Z =   109.147  mm,
	W =    41.080 deg,	P =   -17.089 deg,	R =    29.592 deg
   GP2:
	UF : 1, UT : 1,
	J1=    90.000 deg,	J2=   -90.000 deg
};
P[522]{
   GP1:
	UF : 1, UT : 1,		CONFIG : 'N U T, 0, 0, 0',
	X =  2502.595  mm,	Y =   166.392  mm,	Z =   -10.256  mm,
	W =    37.875 deg,	P =   -26.388 deg,	R =    31.559 deg
   GP2:
	UF : 1, UT : 1,
	J1=    90.000 deg,	J2=   -90.000 deg
};
P[523]{
   GP1:
	UF : 1, UT : 1,		CONFIG : 'N U T, 0, 0, 0',
	X =  2457.453  mm,	Y =   167.249  mm,	Z =   -10.255  mm,
	W =    37.875 deg,	P =   -26.388 deg,	R =    31.559 deg
   GP2:
	UF : 1, UT : 1,
	J1=    90.000 deg,	J2=   -90.000 deg
};
P[524]{
   GP1:
	UF : 1, UT : 1,		CONFIG : 'N U T, 0, 0, 0',
	X =  2438.969  mm,	Y =   167.503  mm,	Z =    -9.377  mm,
	W =    43.420 deg,	P =   -13.215 deg,	R =    37.757 deg
   GP2:
	UF : 1, UT : 1,
	J1=    90.000 deg,	J2=   -90.000 deg
};
P[525]{
   GP1:
	UF : 1, UT : 1,		CONFIG : 'N U T, 0, 0, 0',
	X =  2340.804  mm,	Y =    96.102  mm,	Z =    56.984  mm,
	W =    34.887 deg,	P =   -26.988 deg,	R =    21.909 deg
   GP2:
	UF : 1, UT : 1,
	J1=    90.000 deg,	J2=   -90.000 deg
};
P[526]{
   GP1:
	UF : 1, UT : 1,		CONFIG : 'N U T, 0, 0, 0',
	X =  2334.769  mm,	Y =  -176.256  mm,	Z =   129.823  mm,
	W =    49.996 deg,	P =    12.253 deg,	R =   -42.841 deg
   GP2:
	UF : 1, UT : 1,
	J1=    90.000 deg,	J2=   -90.000 deg
};
P[527]{
   GP1:
	UF : 1, UT : 1,		CONFIG : 'N U T, 0, 0, 0',
	X =  1274.769  mm,	Y =  -176.256  mm,	Z =   129.823  mm,
	W =    14.633 deg,	P =    39.206 deg,	R =   -59.040 deg
   GP2:
	UF : 1, UT : 1,
	J1=    90.000 deg,	J2=   -90.000 deg
};
P[528]{
   GP1:
	UF : 1, UT : 1,		CONFIG : 'N U T, 0, 0, 0',
	X =  1137.626  mm,	Y =   231.744  mm,	Z =   129.823  mm,
	W =     5.452 deg,	P =    45.384 deg,	R =    96.559 deg
   GP2:
	UF : 1, UT : 1,
	J1=    90.000 deg,	J2=   -90.000 deg
};
P[529]{
   GP1:
	UF : 1, UT : 1,		CONFIG : 'N U T, 0, 0, 0',
	X =  1702.626  mm,	Y =   216.744  mm,	Z =    45.395  mm,
	W =   -35.057 deg,	P =    31.336 deg,	R =    18.229 deg
   GP2:
	UF : 1, UT : 1,
	J1=    90.000 deg,	J2=   -90.000 deg
};
P[530]{
   GP1:
	UF : 1, UT : 1,		CONFIG : 'N U T, 0, 0, 0',
	X =  1681.437  mm,	Y =   -64.027  mm,	Z =   -18.046  mm,
	W =    41.392 deg,	P =    19.514 deg,	R =   -17.203 deg
   GP2:
	UF : 1, UT : 1,
	J1=    90.000 deg,	J2=   -90.000 deg
};
P[531]{
   GP1:
	UF : 1, UT : 1,		CONFIG : 'N U T, 0, 0, 0',
	X =  1641.116  mm,	Y =   -63.889  mm,	Z =   -17.838  mm,
	W =    41.393 deg,	P =    19.514 deg,	R =   -16.107 deg
   GP2:
	UF : 1, UT : 1,
	J1=    90.000 deg,	J2=   -90.000 deg
};
P[532]{
   GP1:
	UF : 1, UT : 1,		CONFIG : 'N U T, 0, 0, 0',
	X =  1633.330  mm,	Y =   -64.104  mm,	Z =   -17.838  mm,
	W =    41.392 deg,	P =    19.514 deg,	R =     3.473 deg
   GP2:
	UF : 1, UT : 1,
	J1=    90.000 deg,	J2=   -90.000 deg
};
P[533]{
   GP1:
	UF : 1, UT : 1,		CONFIG : 'N U T, 0, 0, 0',
	X =  1625.901  mm,	Y =   -70.389  mm,	Z =   -17.839  mm,
	W =    41.392 deg,	P =    19.514 deg,	R =    24.112 deg
   GP2:
	UF : 1, UT : 1,
	J1=    90.000 deg,	J2=   -90.000 deg
};
P[534]{
   GP1:
	UF : 1, UT : 1,		CONFIG : 'N U T, 0, 0, 0',
	X =  1968.756  mm,	Y =   235.799  mm,	Z =    41.294  mm,
	W =   -37.049 deg,	P =    22.562 deg,	R =    41.911 deg
   GP2:
	UF : 1, UT : 1,
	J1=    90.000 deg,	J2=   -90.000 deg
};
P[535]{
   GP1:
	UF : 1, UT : 1,		CONFIG : 'N U T, 0, 0, 0',
	X =  2281.156  mm,	Y =   263.463  mm,	Z =    29.688  mm,
	W =   -37.041 deg,	P =    22.569 deg,	R =    41.916 deg
   GP2:
	UF : 1, UT : 1,
	J1=    83.000 deg,	J2=   -90.000 deg
};
P[536]{
   GP1:
	UF : 1, UT : 1,		CONFIG : 'N U T, 0, 0, 0',
	X =  2487.498  mm,	Y =   206.111  mm,	Z =    13.958  mm,
	W =   -43.230 deg,	P =      .800 deg,	R =   -58.961 deg
   GP2:
	UF : 1, UT : 1,
	J1=    83.000 deg,	J2=   -90.000 deg
};
P[537]{
   GP1:
	UF : 1, UT : 1,		CONFIG : 'N U T, 0, 0, 0',
	X =  2487.758  mm,	Y =   132.800  mm,	Z =    41.293  mm,
	W =   -42.488 deg,	P =     1.841 deg,	R =   -72.344 deg
   GP2:
	UF : 1, UT : 1,
	J1=    83.000 deg,	J2=   -90.000 deg
};
P[538]{
   GP1:
	UF : 1, UT : 1,		CONFIG : 'N U T, 0, 0, 0',
	X =  1598.660  mm,	Y =   -98.510  mm,	Z =   -16.821  mm,
	W =    37.029 deg,	P =    27.659 deg,	R =    15.297 deg
   GP2:
	UF : 1, UT : 1,
	J1=    90.000 deg,	J2=   -90.000 deg
};
P[539]{
   GP1:
	UF : 1, UT : 1,		CONFIG : 'N U T, 0, 0, 0',
	X =  1578.869  mm,	Y =  -108.243  mm,	Z =   -16.384  mm,
	W =    38.940 deg,	P =    23.604 deg,	R =   -29.723 deg
   GP2:
	UF : 1, UT : 1,
	J1=    90.000 deg,	J2=   -90.000 deg
};
P[540]{
   GP1:
	UF : 1, UT : 1,		CONFIG : 'N U T, 0, 0, 0',
	X =  1554.046  mm,	Y =   -82.166  mm,	Z =   -15.888  mm,
	W =    36.731 deg,	P =    28.082 deg,	R =  -117.245 deg
   GP2:
	UF : 1, UT : 1,
	J1=    90.000 deg,	J2=   -90.000 deg
};
P[541]{
   GP1:
	UF : 1, UT : 1,		CONFIG : 'N U T, 0, 0, 0',
	X =  1550.331  mm,	Y =   -39.595  mm,	Z =   -15.888  mm,
	W =    36.731 deg,	P =    28.082 deg,	R =  -114.509 deg
   GP2:
	UF : 1, UT : 1,
	J1=    90.000 deg,	J2=   -90.000 deg
};
P[542]{
   GP1:
	UF : 1, UT : 1,		CONFIG : 'N U T, 0, 0, 0',
	X =  2487.758  mm,	Y =   132.800  mm,	Z =    41.293  mm,
	W =   -42.488 deg,	P =     1.841 deg,	R =   -72.344 deg
   GP2:
	UF : 1, UT : 1,
	J1=    83.000 deg,	J2=   -90.000 deg
};
P[543]{
   GP1:
	UF : 1, UT : 1,		CONFIG : 'N U T, 0, 0, 0',
	X =  2487.757  mm,	Y =   235.800  mm,	Z =    41.293  mm,
	W =   -46.494 deg,	P =   -14.946 deg,	R =     1.465 deg
   GP2:
	UF : 1, UT : 1,
	J1=    83.000 deg,	J2=   -90.000 deg
};
P[544]{
   GP1:
	UF : 1, UT : 1,		CONFIG : 'N U T, 0, 0, 0',
	X =  2363.757  mm,	Y =   235.799  mm,	Z =    47.485  mm,
	W =   -46.494 deg,	P =   -14.946 deg,	R =     1.465 deg
   GP2:
	UF : 1, UT : 1,
	J1=    90.000 deg,	J2=   -90.000 deg
};
P[545]{
   GP1:
	UF : 1, UT : 1,		CONFIG : 'N U T, 0, 0, 0',
	X =  1550.258  mm,	Y =   -32.023  mm,	Z =   -15.889  mm,
	W =    36.731 deg,	P =    28.082 deg,	R =   -80.640 deg
   GP2:
	UF : 1, UT : 1,
	J1=    90.000 deg,	J2=   -90.000 deg
};
P[546]{
   GP1:
	UF : 1, UT : 1,		CONFIG : 'N U T, 0, 0, 0',
	X =  1542.901  mm,	Y =   -27.523  mm,	Z =   -15.890  mm,
	W =    36.730 deg,	P =    28.082 deg,	R =   -43.974 deg
   GP2:
	UF : 1, UT : 1,
	J1=    90.000 deg,	J2=   -90.000 deg
};
P[547]{
   GP1:
	UF : 1, UT : 1,		CONFIG : 'N U T, 0, 0, 0',
	X =  2483.422  mm,	Y =   242.950  mm,	Z =    62.981  mm,
	W =   -44.990 deg,	P =    -1.038 deg,	R =    17.559 deg
   GP2:
	UF : 1, UT : 1,
	J1=    90.000 deg,	J2=   -90.000 deg
};
P[548]{
   GP1:
	UF : 1, UT : 1,		CONFIG : 'N U T, 0, 0, 0',
	X =  2280.422  mm,	Y =   242.950  mm,	Z =    62.981  mm,
	W =   -44.990 deg,	P =    -1.038 deg,	R =    17.559 deg
   GP2:
	UF : 1, UT : 1,
	J1=    90.000 deg,	J2=   -90.000 deg
};
P[549]{
   GP1:
	UF : 1, UT : 1,		CONFIG : 'N U T, 0, 0, 0',
	X =  2280.422  mm,	Y =   142.950  mm,	Z =    62.981  mm,
	W =   -44.990 deg,	P =    -1.038 deg,	R =    17.559 deg
   GP2:
	UF : 1, UT : 1,
	J1=    90.000 deg,	J2=   -90.000 deg
};
P[550]{
   GP1:
	UF : 1, UT : 1,		CONFIG : 'N U T, 0, 0, 0',
	X =  1537.073  mm,	Y =   -25.152  mm,	Z =   -15.489  mm,
	W =    37.435 deg,	P =    27.430 deg,	R =   -47.498 deg
   GP2:
	UF : 1, UT : 1,
	J1=    90.000 deg,	J2=   -90.000 deg
};
P[551]{
   GP1:
	UF : 1, UT : 1,		CONFIG : 'N U T, 0, 0, 0',
	X =  2355.837  mm,	Y =   167.626  mm,	Z =   -10.411  mm,
	W =    38.116 deg,	P =   -25.970 deg,	R =    27.303 deg
   GP2:
	UF : 1, UT : 1,
	J1=    90.000 deg,	J2=   -90.000 deg
};
P[552]{
   GP1:
	UF : 1, UT : 1,		CONFIG : 'N U T, 0, 0, 0',
	X =  2398.766  mm,	Y =   167.626  mm,	Z =   -10.411  mm,
	W =    38.116 deg,	P =   -25.970 deg,	R =    27.303 deg
   GP2:
	UF : 1, UT : 1,
	J1=    90.000 deg,	J2=   -90.000 deg
};
P[553]{
   GP1:
	UF : 1, UT : 1,		CONFIG : 'N U T, 0, 0, 0',
	X =  2280.422  mm,	Y =   218.557  mm,	Z =   105.269  mm,
	W =   -44.990 deg,	P =    -1.038 deg,	R =    25.270 deg
   GP2:
	UF : 1, UT : 1,
	J1=    90.000 deg,	J2=   -90.000 deg
};
P[554]{
   GP1:
	UF : 1, UT : 1,		CONFIG : 'N U T, 0, 0, 0',
	X =  1204.422  mm,	Y =   218.557  mm,	Z =   105.269  mm,
	W =   -29.046 deg,	P =    29.449 deg,	R =    29.350 deg
   GP2:
	UF : 1, UT : 1,
	J1=    90.000 deg,	J2=   -90.000 deg
};
P[555]{
   GP1:
	UF : 1, UT : 1,		CONFIG : 'N U T, 0, 0, 0',
	X =  1204.422  mm,	Y =  -167.443  mm,	Z =  1122.269  mm,
	W =   -44.990 deg,	P =    -1.038 deg,	R =    25.270 deg
   GP2:
	UF : 1, UT : 1,
	J1=    90.000 deg,	J2=   -90.000 deg
};
P[556]{
   GP1:
	UF : 1, UT : 1,		CONFIG : 'N U T, 0, 0, 0',
	X =  2328.690  mm,	Y =   -25.109  mm,	Z =   925.961  mm,
	W =    38.029 deg,	P =    27.224 deg,	R =   -32.413 deg
   GP2:
	UF : 1, UT : 1,
	J1=    90.000 deg,	J2=   -90.000 deg
};
P[557]{
   GP1:
	UF : 1, UT : 1,		CONFIG : 'N U T, 0, 0, 0',
	X =  2417.510  mm,	Y =   166.863  mm,	Z =    -9.646  mm,
	W =    15.651 deg,	P =   -37.247 deg,	R =    40.103 deg
   GP2:
	UF : 1, UT : 1,
	J1=    89.989 deg,	J2=   -90.001 deg
};
P[558]{
   GP1:
	UF : 1, UT : 1,		CONFIG : 'N U T, 0, 0, 0',
	X =  1662.158  mm,	Y =   194.594  mm,	Z =   -16.054  mm,
	W =   -37.043 deg,	P =    22.560 deg,	R =   -17.134 deg
   GP2:
	UF : 1, UT : 1,
	J1=    90.000 deg,	J2=   -90.000 deg
};
P[559]{
   GP1:
	UF : 1, UT : 1,		CONFIG : 'N U T, 0, 0, 0',
	X =  2407.814  mm,	Y =    -3.230  mm,	Z =   914.873  mm,
	W =    36.706 deg,	P =    26.470 deg,	R =   -16.230 deg
   GP2:
	UF : 1, UT : 1,
	J1=    90.000 deg,	J2=   -90.000 deg
};
P[560]{
   GP1:
	UF : 1, UT : 1,		CONFIG : 'N U T, 0, 0, 0',
	X =  2432.823  mm,	Y =   104.215  mm,	Z =   863.805  mm,
	W =     4.851 deg,	P =    34.958 deg,	R =    24.131 deg
   GP2:
	UF : 1, UT : 1,
	J1=    89.999 deg,	J2=   -90.000 deg
};
P[561]{
   GP1:
	UF : 1, UT : 1,		CONFIG : 'N U T, 0, 0, 0',
	X =  1697.928  mm,	Y =   193.618  mm,	Z =   -16.152  mm,
	W =   -37.049 deg,	P =    22.568 deg,	R =    34.048 deg
   GP2:
	UF : 1, UT : 1,
	J1=    90.000 deg,	J2=   -90.000 deg
};
P[562]{
   GP1:
	UF : 1, UT : 1,		CONFIG : 'N U T, 0, 0, 0',
	X =  1965.748  mm,	Y =   191.443  mm,	Z =   -19.982  mm,
	W =   -37.049 deg,	P =    22.562 deg,	R =    34.049 deg
   GP2:
	UF : 1, UT : 1,
	J1=    90.000 deg,	J2=   -90.000 deg
};
P[563]{
   GP1:
	UF : 1, UT : 1,		CONFIG : 'N U T, 0, 0, 0',
	X =  2459.632  mm,	Y =   122.370  mm,	Z =   906.747  mm,
	W =    -6.207 deg,	P =    17.663 deg,	R =    19.082 deg
   GP2:
	UF : 1, UT : 1,
	J1=    89.999 deg,	J2=   -90.000 deg
};
P[564]{
   GP1:
	UF : 1, UT : 1,		CONFIG : 'N U T, 0, 0, 0',
	X =  1677.456  mm,	Y = -1378.259  mm,	Z =  1040.445  mm,
	W =   -45.493 deg,	P =   -19.537 deg,	R =    48.719 deg
   GP2:
	UF : 1, UT : 1,
	J1=   180.000 deg,	J2=  -125.000 deg
};
P[565]{
   GP1:
	UF : 1, UT : 1,		CONFIG : 'N U T, 0, 0, 0',
	X =  2301.523  mm,	Y =   100.306  mm,	Z =   896.809  mm,
	W =   -38.032 deg,	P =    -5.730 deg,	R =    38.955 deg
   GP2:
	UF : 1, UT : 1,
	J1=    89.999 deg,	J2=   -90.000 deg
};
P[566]{
   GP1:
	UF : 1, UT : 1,		CONFIG : 'N U T, 0, 0, 0',
	X =  1988.238  mm,	Y =   192.885  mm,	Z =   -18.010  mm,
	W =   -37.043 deg,	P =    22.566 deg,	R =    68.908 deg
   GP2:
	UF : 1, UT : 1,
	J1=    90.000 deg,	J2=   -90.000 deg
};
P[567]{
   GP1:
	UF : 1, UT : 1,		CONFIG : 'N U T, 0, 0, 0',
	X =  2384.746  mm,	Y =    82.939  mm,	Z =   -23.139  mm,
	W =   -47.989 deg,	P =     7.880 deg,	R =   -47.839 deg
   GP2:
	UF : 1, UT : 1,
	J1=    83.000 deg,	J2=   -90.000 deg
};
P[568]{
   GP1:
	UF : 1, UT : 1,		CONFIG : 'N U T, 0, 0, 0',
	X =  2343.829  mm,	Y =   125.019  mm,	Z =   873.736  mm,
	W =   -38.032 deg,	P =    -5.730 deg,	R =    38.955 deg
   GP2:
	UF : 1, UT : 1,
	J1=    89.999 deg,	J2=   -90.000 deg
};
P[569]{
   GP1:
	UF : 1, UT : 1,		CONFIG : 'N U T, 0, 0, 0',
	X =  1695.422  mm,	Y =   -78.871  mm,	Z =  1381.555  mm,
	W =    -4.515 deg,	P =      .965 deg,	R =    -2.729 deg
   GP2:
	UF : 1, UT : 1,
	J1=    90.000 deg,	J2=   -90.000 deg
};
P[570]{
   GP1:
	UF : 1, UT : 1,		CONFIG : 'N U T, 0, 0, 0',
	X =  2545.769  mm,	Y =   814.952  mm,	Z =   -71.983  mm,
	W =   -32.484 deg,	P =     1.246 deg,	R =    91.954 deg
   GP2:
	UF : 1, UT : 1,
	J1=    80.000 deg,	J2=   -90.000 deg
};
P[571]{
   GP1:
	UF : 1, UT : 1,		CONFIG : 'N U T, 0, 0, 0',
	X =  1618.043  mm,	Y = -1395.782  mm,	Z =  1053.900  mm,
	W =   -44.560 deg,	P =   -18.266 deg,	R =    45.822 deg
   GP2:
	UF : 1, UT : 1,
	J1=   180.000 deg,	J2=  -125.000 deg
};
P[572]{
   GP1:
	UF : 1, UT : 1,		CONFIG : 'N U T, 0, 0, 0',
	X =  2106.244  mm,	Y =  -177.973  mm,	Z =   164.824  mm,
	W =    -4.184 deg,	P =     7.592 deg,	R =    43.674 deg
   GP2:
	UF : 1, UT : 1,
	J1=    90.000 deg,	J2=  -100.000 deg
};
P[573]{
   GP1:
	UF : 1, UT : 1,		CONFIG : 'N U T, 0, 0, 0',
	X =  2106.243  mm,	Y =   -20.258  mm,	Z =   164.824  mm,
	W =     2.218 deg,	P =    14.051 deg,	R =    70.281 deg
   GP2:
	UF : 1, UT : 1,
	J1=    90.000 deg,	J2=  -100.000 deg
};
P[574]{
   GP1:
	UF : 1, UT : 1,		CONFIG : 'N U T, 0, 0, 0',
	X =  2383.889  mm,	Y =    97.654  mm,	Z =   -23.139  mm,
	W =   -47.989 deg,	P =     7.880 deg,	R =   -71.350 deg
   GP2:
	UF : 1, UT : 1,
	J1=    83.000 deg,	J2=   -90.000 deg
};
P[575]{
   GP1:
	UF : 1, UT : 1,		CONFIG : 'N U T, 0, 0, 0',
	X =  2383.891  mm,	Y =   140.297  mm,	Z =   -23.140  mm,
	W =   -47.989 deg,	P =     7.880 deg,	R =   -71.350 deg
   GP2:
	UF : 1, UT : 1,
	J1=    83.000 deg,	J2=   -90.000 deg
};
P[576]{
   GP1:
	UF : 1, UT : 1,		CONFIG : 'N U T, 0, 0, 0',
	X =  2113.743  mm,	Y =   -23.258  mm,	Z =   164.824  mm,
	W =     2.218 deg,	P =    14.051 deg,	R =    70.281 deg
   GP2:
	UF : 1, UT : 1,
	J1=    90.000 deg,	J2=  -100.000 deg
};
P[577]{
   GP1:
	UF : 1, UT : 1,		CONFIG : 'N U T, 0, 0, 0',
	X =  2106.244  mm,	Y =  -177.973  mm,	Z =   164.824  mm,
	W =    -4.184 deg,	P =     7.592 deg,	R =    43.674 deg
   GP2:
	UF : 1, UT : 1,
	J1=    90.000 deg,	J2=  -100.000 deg
};
P[578]{
   GP1:
	UF : 1, UT : 1,		CONFIG : 'N U T, 0, 0, 0',
	X =  2154.661  mm,	Y =  -177.973  mm,	Z =   164.824  mm,
	W =    28.994 deg,	P =   -15.433 deg,	R =    30.441 deg
   GP2:
	UF : 1, UT : 1,
	J1=    90.000 deg,	J2=   -90.000 deg
};
P[579]{
   GP1:
	UF : 1, UT : 1,		CONFIG : 'N U T, 0, 0, 0',
	X =  2383.459  mm,	Y =   165.155  mm,	Z =   -23.142  mm,
	W =   -47.988 deg,	P =     7.880 deg,	R =  -106.126 deg
   GP2:
	UF : 1, UT : 1,
	J1=    83.000 deg,	J2=   -90.000 deg
};
P[580]{
   GP1:
	UF : 1, UT : 1,		CONFIG : 'N U T, 0, 0, 0',
	X =  2356.304  mm,	Y =   178.504  mm,	Z =   -10.428  mm,
	W =   -44.818 deg,	P =    -4.562 deg,	R =    -2.490 deg
   GP2:
	UF : 1, UT : 1,
	J1=    90.000 deg,	J2=   -90.000 deg
};
P[581]{
   GP1:
	UF : 1, UT : 1,		CONFIG : 'N U T, 0, 0, 0',
	X =  2158.527  mm,	Y =  -106.081  mm,	Z =    42.026  mm,
	W =    44.885 deg,	P =     3.628 deg,	R =    -3.635 deg
   GP2:
	UF : 1, UT : 1,
	J1=    90.000 deg,	J2=   -90.000 deg
};
P[582]{
   GP1:
	UF : 1, UT : 1,		CONFIG : 'N U T, 0, 0, 0',
	X =  2501.518  mm,	Y =   177.433  mm,	Z =   -10.428  mm,
	W =   -44.818 deg,	P =    -4.562 deg,	R =    -2.490 deg
   GP2:
	UF : 1, UT : 1,
	J1=    90.000 deg,	J2=   -90.000 deg
};
P[583]{
   GP1:
	UF : 1, UT : 1,		CONFIG : 'N U T, 0, 0, 0',
	X =  2355.927  mm,	Y =    83.611  mm,	Z =   -11.600  mm,
	W =   -44.391 deg,	P =     8.269 deg,	R =    10.730 deg
   GP2:
	UF : 1, UT : 1,
	J1=    90.000 deg,	J2=   -90.000 deg
};
P[584]{
   GP1:
	UF : 1, UT : 1,		CONFIG : 'N U T, 0, 0, 0',
	X =  2401.784  mm,	Y =    82.111  mm,	Z =   -11.600  mm,
	W =   -44.391 deg,	P =     8.269 deg,	R =    12.650 deg
   GP2:
	UF : 1, UT : 1,
	J1=    90.000 deg,	J2=   -90.000 deg
};
P[585]{
   GP1:
	UF : 1, UT : 1,		CONFIG : 'N U T, 0, 0, 0',
	X =  2060.197  mm,	Y =  -106.080  mm,	Z =    42.026  mm,
	W =    44.885 deg,	P =     3.628 deg,	R =    -3.635 deg
   GP2:
	UF : 1, UT : 1,
	J1=    90.000 deg,	J2=   -90.000 deg
};
P[586]{
   GP1:
	UF : 1, UT : 1,		CONFIG : 'N U T, 0, 0, 0',
	X =  2415.080  mm,	Y =    90.438  mm,	Z =    -4.548  mm,
	W =   -44.382 deg,	P =     8.277 deg,	R =    40.042 deg
   GP2:
	UF : 1, UT : 1,
	J1=    90.000 deg,	J2=   -90.000 deg
};
P[587]{
   GP1:
	UF : 1, UT : 1,		CONFIG : 'N U T, 0, 0, 0',
	X =  2340.827  mm,	Y =    56.155  mm,	Z =   838.039  mm,
	W =    38.029 deg,	P =    27.224 deg,	R =   -32.413 deg
   GP2:
	UF : 1, UT : 1,
	J1=    90.000 deg,	J2=   -90.000 deg
};
P[588]{
   GP1:
	UF : 1, UT : 1,		CONFIG : 'N U T, 0, 0, 0',
	X =  2406.112  mm,	Y =    90.298  mm,	Z =   838.040  mm,
	W =    38.029 deg,	P =    27.224 deg,	R =   -32.413 deg
   GP2:
	UF : 1, UT : 1,
	J1=    90.000 deg,	J2=   -90.000 deg
};
P[589]{
   GP1:
	UF : 1, UT : 1,		CONFIG : 'N U T, 0, 0, 0',
	X =  1890.253  mm,	Y =  -197.333  mm,	Z =   104.046  mm,
	W =    40.690 deg,	P =   -21.162 deg,	R =    -6.795 deg
   GP2:
	UF : 1, UT : 1,
	J1=    90.000 deg,	J2=   -90.000 deg
};
P[590]{
   GP1:
	UF : 1, UT : 1,		CONFIG : 'N U T, 0, 0, 0',
	X =  1890.254  mm,	Y =  -197.333  mm,	Z =   104.046  mm,
	W =   -33.760 deg,	P =   -16.746 deg,	R =    41.760 deg
   GP2:
	UF : 1, UT : 1,
	J1=    90.000 deg,	J2=   -90.000 deg
};
P[591]{
   GP1:
	UF : 1, UT : 1,		CONFIG : 'N U T, 0, 0, 0',
	X =  2024.254  mm,	Y =  -116.333  mm,	Z =   104.046  mm,
	W =   -36.632 deg,	P =    -7.222 deg,	R =    55.482 deg
   GP2:
	UF : 1, UT : 1,
	J1=    90.000 deg,	J2=   -90.000 deg
};
P[592]{
   GP1:
	UF : 1, UT : 1,		CONFIG : 'N U T, 0, 0, 0',
	X =  2396.431  mm,	Y =   116.616  mm,	Z =   834.888  mm,
	W =     5.388 deg,	P =    42.666 deg,	R =    25.064 deg
   GP2:
	UF : 1, UT : 1,
	J1=    89.999 deg,	J2=   -90.000 deg
};
P[593]{
   GP1:
	UF : 1, UT : 1,		CONFIG : 'N U T, 0, 0, 0',
	X =  2326.230  mm,	Y =    84.543  mm,	Z =   839.612  mm,
	W =   -38.032 deg,	P =    -5.730 deg,	R =    38.955 deg
   GP2:
	UF : 1, UT : 1,
	J1=    89.999 deg,	J2=   -90.000 deg
};
P[594]{
   GP1:
	UF : 1, UT : 1,		CONFIG : 'N U T, 0, 0, 0',
	X =  2390.516  mm,	Y =   118.971  mm,	Z =   839.612  mm,
	W =   -38.032 deg,	P =    -5.730 deg,	R =    38.955 deg
   GP2:
	UF : 1, UT : 1,
	J1=    89.999 deg,	J2=   -90.000 deg
};
P[595]{
   GP1:
	UF : 1, UT : 1,		CONFIG : 'N U T, 0, 0, 0',
	X =  2056.301  mm,	Y =   -98.366  mm,	Z =    49.506  mm,
	W =   -42.382 deg,	P =     2.305 deg,	R =   105.198 deg
   GP2:
	UF : 1, UT : 1,
	J1=    90.000 deg,	J2=   -90.000 deg
};
P[596]{
   GP1:
	UF : 1, UT : 1,		CONFIG : 'N U T, 0, 0, 1',
	X =  1663.323  mm,	Y =  -387.368  mm,	Z =   408.939  mm,
	W =   -27.547 deg,	P =    30.353 deg,	R =   152.229 deg
   GP2:
	UF : 1, UT : 1,
	J1=    90.000 deg,	J2=   -90.000 deg
};
P[597]{
   GP1:
	UF : 1, UT : 1,		CONFIG : 'N U T, 0, 0, 1',
	X =  1656.330  mm,	Y =  -300.541  mm,	Z =  1123.310  mm,
	W =    -9.281 deg,	P =    48.130 deg,	R =  -175.012 deg
   GP2:
	UF : 1, UT : 1,
	J1=    90.000 deg,	J2=   -90.000 deg
};
P[598]{
   GP1:
	UF : 1, UT : 1,		CONFIG : 'N U T, 0, 0, 1',
	X =  2106.086  mm,	Y =  -147.825  mm,	Z =   986.847  mm,
	W =    -2.744 deg,	P =    30.268 deg,	R =  -167.022 deg
   GP2:
	UF : 1, UT : 1,
	J1=    90.000 deg,	J2=   -90.000 deg
};
P[599]{
   GP1:
	UF : 1, UT : 1,		CONFIG : 'N U T, 0, 0, 0',
	X =  2556.458  mm,	Y =   802.225  mm,	Z =   -73.705  mm,
	W =   -29.311 deg,	P =   -14.722 deg,	R =   104.314 deg
   GP2:
	UF : 1, UT : 1,
	J1=    80.000 deg,	J2=   -90.000 deg
};
P[600]{
   GP1:
	UF : 1, UT : 1,		CONFIG : 'N U T, 0, 0, 0',
	X =  2004.590  mm,	Y =   -97.008  mm,	Z =    -9.937  mm,
	W =    40.372 deg,	P =    23.930 deg,	R =    74.347 deg
   GP2:
	UF : 1, UT : 1,
	J1=    90.000 deg,	J2=  -100.000 deg
};
P[601]{
   GP1:
	UF : 1, UT : 1,		CONFIG : 'N U T, 0, 0, 0',
	X =  2003.703  mm,	Y =   128.202  mm,	Z =   -49.382  mm,
	W =    45.687 deg,	P =     4.511 deg,	R =    78.829 deg
   GP2:
	UF : 1, UT : 1,
	J1=    90.000 deg,	J2=  -100.000 deg
};
P[602]{
   GP1:
	UF : 1, UT : 1,		CONFIG : 'N U T, 0, 0, 0',
	X =  2224.724  mm,	Y =   -63.982  mm,	Z =    -4.139  mm,
	W =    44.897 deg,	P =    -3.424 deg,	R =     3.430 deg
   GP2:
	UF : 1, UT : 1,
	J1=    90.000 deg,	J2=   -90.000 deg
};
P[603]{
   GP1:
	UF : 1, UT : 1,		CONFIG : 'N U T, 0, 0, 0',
	X =  2255.938  mm,	Y =   -63.982  mm,	Z =    -4.139  mm,
	W =    44.897 deg,	P =    -3.424 deg,	R =     3.430 deg
   GP2:
	UF : 1, UT : 1,
	J1=    90.000 deg,	J2=   -90.000 deg
};
P[604]{
   GP1:
	UF : 1, UT : 1,		CONFIG : 'N U T, 0, 0, 0',
	X =  2129.118  mm,	Y =   -62.477  mm,	Z =   -12.526  mm,
	W =    44.886 deg,	P =     3.630 deg,	R =    -4.912 deg
   GP2:
	UF : 1, UT : 1,
	J1=    90.000 deg,	J2=   -90.000 deg
};
P[605]{
   GP1:
	UF : 1, UT : 1,		CONFIG : 'N U T, 0, 0, 0',
	X =  2197.333  mm,	Y =   -62.477  mm,	Z =   -12.526  mm,
	W =    44.886 deg,	P =     3.630 deg,	R =    -4.912 deg
   GP2:
	UF : 1, UT : 1,
	J1=    90.000 deg,	J2=   -90.000 deg
};
P[606]{
   GP1:
	UF : 1, UT : 1,		CONFIG : 'N U T, 0, 0, 0',
	X =  2206.333  mm,	Y =   -63.120  mm,	Z =   -12.525  mm,
	W =    44.886 deg,	P =     3.630 deg,	R =   -13.666 deg
   GP2:
	UF : 1, UT : 1,
	J1=    90.000 deg,	J2=   -90.000 deg
};
P[607]{
   GP1:
	UF : 1, UT : 1,		CONFIG : 'N U T, 0, 0, 0',
	X =  2096.605  mm,	Y =  -181.583  mm,	Z =   897.867  mm,
	W =     -.064 deg,	P =    31.734 deg,	R =  -164.129 deg
   GP2:
	UF : 1, UT : 1,
	J1=    90.000 deg,	J2=   -90.000 deg
};
P[608]{
   GP1:
	UF : 1, UT : 1,		CONFIG : 'N U T, 0, 0, 0',
	X =  2114.149  mm,	Y =  -253.336  mm,	Z =   921.197  mm,
	W =     1.157 deg,	P =    35.359 deg,	R =   -90.786 deg
   GP2:
	UF : 1, UT : 1,
	J1=    90.000 deg,	J2=   -90.000 deg
};
P[609]{
   GP1:
	UF : 1, UT : 1,		CONFIG : 'N U T, 0, 0, 0',
	X =  1983.423  mm,	Y =   -63.309  mm,	Z =   -19.831  mm,
	W =    44.885 deg,	P =     3.628 deg,	R =    -8.844 deg
   GP2:
	UF : 1, UT : 1,
	J1=    90.000 deg,	J2=   -90.000 deg
};
P[610]{
   GP1:
	UF : 1, UT : 1,		CONFIG : 'N U T, 0, 0, 0',
	X =  2098.137  mm,	Y =   -63.523  mm,	Z =   -20.045  mm,
	W =    44.885 deg,	P =     3.628 deg,	R =   -12.185 deg
   GP2:
	UF : 1, UT : 1,
	J1=    90.000 deg,	J2=   -90.000 deg
};
P[611]{
   GP1:
	UF : 1, UT : 1,		CONFIG : 'N U T, 0, 0, 0',
	X =  2107.937  mm,	Y =   -64.825  mm,	Z =   -18.870  mm,
	W =    36.789 deg,	P =   -27.991 deg,	R =    -8.613 deg
   GP2:
	UF : 1, UT : 1,
	J1=    90.000 deg,	J2=   -90.000 deg
};
P[612]{
   GP1:
	UF : 1, UT : 1,		CONFIG : 'N U T, 0, 0, 0',
	X =  2063.279  mm,	Y =  -109.056  mm,	Z =   -13.744  mm,
	W =   -37.498 deg,	P =      .970 deg,	R =    76.656 deg
   GP2:
	UF : 1, UT : 1,
	J1=    90.000 deg,	J2=   -90.000 deg
};
P[613]{
   GP1:
	UF : 1, UT : 1,		CONFIG : 'N U T, 0, 0, 0',
	X =  2087.900  mm,	Y =   -88.864  mm,	Z =   -15.508  mm,
	W =   -37.504 deg,	P =      .973 deg,	R =    76.661 deg
   GP2:
	UF : 1, UT : 1,
	J1=    90.000 deg,	J2=   -90.000 deg
};
P[614]{
   GP1:
	UF : 1, UT : 1,		CONFIG : 'N U T, 0, 0, 0',
	X =  2106.573  mm,	Y =   -68.546  mm,	Z =   -13.129  mm,
	W =   -38.830 deg,	P =     4.264 deg,	R =   105.253 deg
   GP2:
	UF : 1, UT : 1,
	J1=    90.000 deg,	J2=   -90.000 deg
};
P[615]{
   GP1:
	UF : 1, UT : 1,		CONFIG : 'N U T, 0, 0, 1',
	X =  2131.447  mm,	Y =  -156.814  mm,	Z =   826.952  mm,
	W =      .931 deg,	P =    42.959 deg,	R =  -160.609 deg
   GP2:
	UF : 1, UT : 1,
	J1=    90.000 deg,	J2=   -90.000 deg
};
P[616]{
   GP1:
	UF : 1, UT : 1,		CONFIG : 'N U T, 0, 0, 1',
	X =  2139.364  mm,	Y =  -180.053  mm,	Z =   826.306  mm,
	W =      .157 deg,	P =    42.762 deg,	R =  -164.022 deg
   GP2:
	UF : 1, UT : 1,
	J1=    90.000 deg,	J2=   -90.000 deg
};
P[617]{
   GP1:
	UF : 1, UT : 1,		CONFIG : 'N U T, 0, 0, 0',
	X =  2127.920  mm,	Y =  -205.021  mm,	Z =   825.688  mm,
	W =     -.175 deg,	P =    44.066 deg,	R =   109.641 deg
   GP2:
	UF : 1, UT : 1,
	J1=    90.000 deg,	J2=   -90.000 deg
};
P[618]{
   GP1:
	UF : 1, UT : 1,		CONFIG : 'N U T, 0, 0, 0',
	X =  2628.655  mm,	Y =   126.905  mm,	Z =   907.127  mm,
	W =    31.997 deg,	P =    23.849 deg,	R =   -38.788 deg
   GP2:
	UF : 1, UT : 1,
	J1=    90.000 deg,	J2=   -90.000 deg
};
P[619]{
   GP1:
	UF : 1, UT : 1,		CONFIG : 'N U T, 0, 0, 0',
	X =   949.417  mm,	Y =    74.708  mm,	Z =  1003.698  mm,
	W =    14.657 deg,	P =    21.488 deg,	R =   -36.321 deg
   GP2:
	UF : 1, UT : 1,
	J1=    90.000 deg,	J2=   -90.000 deg
};
P[620]{
   GP1:
	UF : 1, UT : 1,		CONFIG : 'N U T, 0, 0, 0',
	X =   931.440  mm,	Y =   198.476  mm,	Z =   335.127  mm,
	W =   -34.527 deg,	P =    19.136 deg,	R =    25.896 deg
   GP2:
	UF : 1, UT : 1,
	J1=    90.000 deg,	J2=   -90.000 deg
};
P[621]{
   GP1:
	UF : 1, UT : 1,		CONFIG : 'N U T, 0, 0, 0',
	X =  1700.688  mm,	Y =   121.333  mm,	Z =   177.127  mm,
	W =   -48.737 deg,	P =     8.784 deg,	R =     7.978 deg
   GP2:
	UF : 1, UT : 1,
	J1=    90.000 deg,	J2=   -90.000 deg
};
P[622]{
   GP1:
	UF : 1, UT : 1,		CONFIG : 'N U T, 0, 0, 0',
	X =  2100.833  mm,	Y =  -196.037  mm,	Z =   827.926  mm,
	W =      .411 deg,	P =    43.126 deg,	R =    21.368 deg
   GP2:
	UF : 1, UT : 1,
	J1=    90.000 deg,	J2=   -90.000 deg
};
P[623]{
   GP1:
	UF : 1, UT : 1,		CONFIG : 'N U T, 0, 0, 0',
	X =  2085.965  mm,	Y =  -148.227  mm,	Z =   828.464  mm,
	W =     -.791 deg,	P =    42.414 deg,	R =    16.379 deg
   GP2:
	UF : 1, UT : 1,
	J1=    90.000 deg,	J2=   -90.000 deg
};
P[624]{
   GP1:
	UF : 1, UT : 1,		CONFIG : 'N U T, 0, 0, 0',
	X =  2104.347  mm,	Y =  -125.535  mm,	Z =   827.812  mm,
	W =      .363 deg,	P =    42.654 deg,	R =   -74.655 deg
   GP2:
	UF : 1, UT : 1,
	J1=    90.000 deg,	J2=   -90.000 deg
};
P[625]{
   GP1:
	UF : 1, UT : 1,		CONFIG : 'N U T, 0, 0, 0',
	X =  2124.774  mm,	Y =  -137.003  mm,	Z =   827.691  mm,
	W =      .919 deg,	P =    43.783 deg,	R =  -158.279 deg
   GP2:
	UF : 1, UT : 1,
	J1=    90.000 deg,	J2=   -90.000 deg
};
P[626]{
   GP1:
	UF : 1, UT : 1,		CONFIG : 'N U T, 0, 0, 0',
	X =  1922.982  mm,	Y =    80.524  mm,	Z =   163.198  mm,
	W =   -51.903 deg,	P =     9.364 deg,	R =    21.482 deg
   GP2:
	UF : 1, UT : 1,
	J1=    90.000 deg,	J2=   -90.000 deg
};
P[627]{
   GP1:
	UF : 1, UT : 1,		CONFIG : 'N U T, 0, 0, 0',
	X =  2179.982  mm,	Y =    80.524  mm,	Z =   163.199  mm,
	W =   -51.227 deg,	P =   -13.564 deg,	R =     3.543 deg
   GP2:
	UF : 1, UT : 1,
	J1=    90.000 deg,	J2=   -90.000 deg
};
P[628]{
   GP1:
	UF : 1, UT : 1,		CONFIG : 'N U T, 0, 0, 0',
	X =  2131.881  mm,	Y =  -155.480  mm,	Z =   826.945  mm,
	W =      .396 deg,	P =    42.883 deg,	R =  -164.093 deg
   GP2:
	UF : 1, UT : 1,
	J1=    89.999 deg,	J2=   -90.000 deg
};
P[629]{
   GP1:
	UF : 1, UT : 1,		CONFIG : 'N U T, 0, 0, 0',
	X =  2104.177  mm,	Y =  -234.400  mm,	Z =   828.213  mm,
	W =     -.450 deg,	P =    39.559 deg,	R =   -90.706 deg
   GP2:
	UF : 1, UT : 1,
	J1=    90.000 deg,	J2=   -90.000 deg
};
P[630]{
   GP1:
	UF : 1, UT : 1,		CONFIG : 'N U T, 0, 0, 0',
	X =  2179.963  mm,	Y =     8.530  mm,	Z =    59.476  mm,
	W =   -44.735 deg,	P =    -5.491 deg,	R =    -5.516 deg
   GP2:
	UF : 1, UT : 1,
	J1=    90.000 deg,	J2=   -90.000 deg
};
P[631]{
   GP1:
	UF : 1, UT : 1,		CONFIG : 'N U T, 0, 0, 0',
	X =  2194.799  mm,	Y =  -234.960  mm,	Z =   828.236  mm,
	W =     -.444 deg,	P =    39.558 deg,	R =   -90.714 deg
   GP2:
	UF : 1, UT : 1,
	J1=    90.000 deg,	J2=   -90.000 deg
};
P[632]{
   GP1:
	UF : 1, UT : 1,		CONFIG : 'N U T, 0, 0, 0',
	X =  2211.805  mm,	Y =  -231.045  mm,	Z =   827.804  mm,
	W =     -.444 deg,	P =    39.559 deg,	R =   -57.817 deg
   GP2:
	UF : 1, UT : 1,
	J1=    90.000 deg,	J2=   -90.000 deg
};
P[633]{
   GP1:
	UF : 1, UT : 1,		CONFIG : 'N U T, 0, 0, 0',
	X =  2221.596  mm,	Y =  -224.020  mm,	Z =   828.211  mm,
	W =     -.441 deg,	P =    39.557 deg,	R =   -44.060 deg
   GP2:
	UF : 1, UT : 1,
	J1=    90.000 deg,	J2=   -90.000 deg
};
P[634]{
   GP1:
	UF : 1, UT : 1,		CONFIG : 'N U T, 0, 0, 0',
	X =  2083.048  mm,	Y =     5.303  mm,	Z =    47.541  mm,
	W =   -44.735 deg,	P =    -5.491 deg,	R =    -5.516 deg
   GP2:
	UF : 1, UT : 1,
	J1=    90.000 deg,	J2=   -90.000 deg
};
P[635]{
   GP1:
	UF : 1, UT : 1,		CONFIG : 'N U T, 0, 0, 0',
	X =  2446.441  mm,	Y =    36.009  mm,	Z =   826.931  mm,
	W =      .118 deg,	P =    42.765 deg,	R =   -42.894 deg
   GP2:
	UF : 1, UT : 1,
	J1=    90.000 deg,	J2=   -90.000 deg
};
P[636]{
   GP1:
	UF : 1, UT : 1,		CONFIG : 'N U T, 0, 0, 0',
	X =  2449.282  mm,	Y =    39.610  mm,	Z =   826.590  mm,
	W =      .108 deg,	P =    42.766 deg,	R =   -49.059 deg
   GP2:
	UF : 1, UT : 1,
	J1=    90.000 deg,	J2=   -90.000 deg
};
P[637]{
   GP1:
	UF : 1, UT : 1,		CONFIG : 'N U T, 0, 0, 0',
	X =  2453.930  mm,	Y =    41.966  mm,	Z =   827.339  mm,
	W =      .113 deg,	P =    42.763 deg,	R =   -56.126 deg
   GP2:
	UF : 1, UT : 1,
	J1=    90.000 deg,	J2=   -90.000 deg
};
P[638]{
   GP1:
	UF : 1, UT : 1,		CONFIG : 'N U T, 0, 0, 0',
	X =  2065.479  mm,	Y =    84.939  mm,	Z =   110.355  mm,
	W =   -44.734 deg,	P =    -5.490 deg,	R =     4.917 deg
   GP2:
	UF : 1, UT : 1,
	J1=    90.000 deg,	J2=   -90.000 deg
};
P[639]{
   GP1:
	UF : 1, UT : 1,		CONFIG : 'N U T, 0, 0, 0',
	X =  1539.706  mm,	Y = -1470.455  mm,	Z =  1071.063  mm,
	W =   -42.856 deg,	P =   -15.293 deg,	R =    39.131 deg
   GP2:
	UF : 1, UT : 1,
	J1=   180.000 deg,	J2=  -125.000 deg
};
P[640]{
   GP1:
	UF : 1, UT : 1,		CONFIG : 'N U T, 0, 0, 0',
	X =  1166.553  mm,	Y = -1374.013  mm,	Z =  1522.225  mm,
	W =   -32.586 deg,	P =   -12.067 deg,	R =    17.529 deg
   GP2:
	UF : 1, UT : 1,
	J1=   180.000 deg,	J2=  -125.000 deg
};
P[641]{
   GP1:
	UF : 1, UT : 1,		CONFIG : 'N U T, 0, 0, 1',
	X =  1608.479  mm,	Y =   191.940  mm,	Z =    59.355  mm,
	W =    36.994 deg,	P =    27.707 deg,	R =  -122.588 deg
   GP2:
	UF : 1, UT : 1,
	J1=    90.000 deg,	J2=   -90.000 deg
};
P[642]{
   GP1:
	UF : 1, UT : 1,		CONFIG : 'N U T, 0, 0, 0',
	X =  2660.076  mm,	Y =   198.015  mm,	Z =   826.173  mm,
	W =    29.495 deg,	P =    29.457 deg,	R =    -6.836 deg
   GP2:
	UF : 1, UT : 1,
	J1=    90.000 deg,	J2=   -90.000 deg
};
P[643]{
   GP1:
	UF : 1, UT : 1,		CONFIG : 'N U T, 0, 0, 0',
	X =  2674.136  mm,	Y =   208.739  mm,	Z =   826.530  mm,
	W =    29.490 deg,	P =    29.462 deg,	R =    -6.842 deg
   GP2:
	UF : 1, UT : 1,
	J1=    90.000 deg,	J2=   -90.000 deg
};
P[644]{
   GP1:
	UF : 1, UT : 1,		CONFIG : 'N U T, 0, 0, 0',
	X =  1960.860  mm,	Y =   -39.301  mm,	Z =    53.624  mm,
	W =   -51.910 deg,	P =     9.369 deg,	R =    25.038 deg
   GP2:
	UF : 1, UT : 1,
	J1=    90.000 deg,	J2=   -90.000 deg
};
P[645]{
   GP1:
	UF : 1, UT : 1,		CONFIG : 'N U T, 0, 0, 0',
	X =  1450.805  mm,	Y =    56.341  mm,	Z =   141.822  mm,
	W =    36.993 deg,	P =    27.706 deg,	R =  -154.189 deg
   GP2:
	UF : 1, UT : 1,
	J1=    90.000 deg,	J2=   -90.000 deg
};
P[646]{
   GP1:
	UF : 1, UT : 1,		CONFIG : 'N U T, 0, 0, 0',
	X =  1476.806  mm,	Y =   169.341  mm,	Z =   386.823  mm,
	W =    23.939 deg,	P =    39.314 deg,	R =  -177.488 deg
   GP2:
	UF : 1, UT : 1,
	J1=    80.000 deg,	J2=   -90.000 deg
};
P[647]{
   GP1:
	UF : 1, UT : 1,		CONFIG : 'N U T, 0, 0, 0',
	X =  2034.807  mm,	Y =   169.341  mm,	Z =   186.823  mm,
	W =    23.939 deg,	P =    39.314 deg,	R =  -177.488 deg
   GP2:
	UF : 1, UT : 1,
	J1=    80.000 deg,	J2=   -90.000 deg
};
P[648]{
   GP1:
	UF : 1, UT : 1,		CONFIG : 'N U T, 0, 0, -1',
	X =  2034.807  mm,	Y =     1.341  mm,	Z =   115.823  mm,
	W =    34.881 deg,	P =    30.459 deg,	R =  -142.693 deg
   GP2:
	UF : 1, UT : 1,
	J1=    80.000 deg,	J2=   -90.000 deg
};
P[649]{
   GP1:
	UF : 1, UT : 1,		CONFIG : 'N U T, 0, 0, 0',
	X =  1938.230  mm,	Y =   -44.353  mm,	Z =    51.798  mm,
	W =   -51.910 deg,	P =     9.369 deg,	R =     4.815 deg
   GP2:
	UF : 1, UT : 1,
	J1=    90.000 deg,	J2=   -90.000 deg
};
P[650]{
   GP1:
	UF : 1, UT : 1,		CONFIG : 'N U T, 0, 0, 0',
	X =  1684.398  mm,	Y =   -47.084  mm,	Z =    53.683  mm,
	W =   -51.917 deg,	P =     9.374 deg,	R =     4.818 deg
   GP2:
	UF : 1, UT : 1,
	J1=    90.000 deg,	J2=   -90.000 deg
};
P[651]{
   GP1:
	UF : 1, UT : 1,		CONFIG : 'N U T, 0, 0, 0',
	X =  1672.627  mm,	Y =   -42.221  mm,	Z =    60.435  mm,
	W =   -51.823 deg,	P =     9.323 deg,	R =   -27.815 deg
   GP2:
	UF : 1, UT : 1,
	J1=    89.996 deg,	J2=   -90.000 deg
};
P[652]{
   GP1:
	UF : 1, UT : 1,		CONFIG : 'N U T, 0, 0, 0',
	X =  2222.567  mm,	Y =   -49.901  mm,	Z =    -4.502  mm,
	W =   -44.735 deg,	P =    -5.491 deg,	R =    -3.611 deg
   GP2:
	UF : 1, UT : 1,
	J1=    90.000 deg,	J2=   -90.000 deg
};
P[653]{
   GP1:
	UF : 1, UT : 1,		CONFIG : 'N U T, 0, 0, 0',
	X =  2258.781  mm,	Y =   -49.901  mm,	Z =    -4.502  mm,
	W =   -44.735 deg,	P =    -5.491 deg,	R =    -3.611 deg
   GP2:
	UF : 1, UT : 1,
	J1=    90.000 deg,	J2=   -90.000 deg
};
P[654]{
   GP1:
	UF : 1, UT : 1,		CONFIG : 'N U T, 0, 0, 0',
	X =  2136.694  mm,	Y =   -48.564  mm,	Z =   -11.246  mm,
	W =   -44.729 deg,	P =    -5.491 deg,	R =    -5.524 deg
   GP2:
	UF : 1, UT : 1,
	J1=    90.000 deg,	J2=   -90.000 deg
};
P[655]{
   GP1:
	UF : 1, UT : 1,		CONFIG : 'N U T, 0, 0, 0',
	X =  2202.479  mm,	Y =   -48.564  mm,	Z =   -11.246  mm,
	W =   -44.729 deg,	P =    -5.491 deg,	R =    -5.524 deg
   GP2:
	UF : 1, UT : 1,
	J1=    90.000 deg,	J2=   -90.000 deg
};
P[656]{
   GP1:
	UF : 1, UT : 1,		CONFIG : 'N U T, 0, 0, 0',
	X =  2207.408  mm,	Y =   -48.565  mm,	Z =   -11.246  mm,
	W =   -44.729 deg,	P =    -5.491 deg,	R =     5.567 deg
   GP2:
	UF : 1, UT : 1,
	J1=    90.000 deg,	J2=   -90.000 deg
};
P[657]{
   GP1:
	UF : 1, UT : 1,		CONFIG : 'N U T, 0, 0, 0',
	X =  2109.643  mm,	Y =   -47.213  mm,	Z =   -18.538  mm,
	W =   -44.735 deg,	P =    -5.490 deg,	R =    -5.516 deg
   GP2:
	UF : 1, UT : 1,
	J1=    90.000 deg,	J2=   -90.000 deg
};
P[658]{
   GP1:
	UF : 1, UT : 1,		CONFIG : 'N U T, 0, 0, 0',
	X =  2025.499  mm,	Y =   -47.428  mm,	Z =   -17.682  mm,
	W =   -44.735 deg,	P =    -5.490 deg,	R =    -5.516 deg
   GP2:
	UF : 1, UT : 1,
	J1=    90.000 deg,	J2=   -90.000 deg
};
P[659]{
   GP1:
	UF : 1, UT : 1,		CONFIG : 'N U T, 0, 0, 0',
	X =  2006.213  mm,	Y =   -49.570  mm,	Z =   -17.896  mm,
	W =   -44.735 deg,	P =    -5.490 deg,	R =   -40.822 deg
   GP2:
	UF : 1, UT : 1,
	J1=    90.000 deg,	J2=   -90.000 deg
};
P[660]{
   GP1:
	UF : 1, UT : 1,		CONFIG : 'N U T, 0, 0, 0',
	X =  1641.471  mm,	Y =   213.113  mm,	Z =   -14.885  mm,
	W =    34.660 deg,	P =    26.416 deg,	R =  -126.988 deg
   GP2:
	UF : 1, UT : 1,
	J1=    89.996 deg,	J2=   -90.000 deg
};
P[661]{
   GP1:
	UF : 1, UT : 1,		CONFIG : 'N U T, 0, 0, 1',
	X =  1643.584  mm,	Y =     6.737  mm,	Z =   -16.612  mm,
	W =    34.637 deg,	P =    26.342 deg,	R =  -123.664 deg
   GP2:
	UF : 1, UT : 1,
	J1=    90.000 deg,	J2=   -90.000 deg
};
P[662]{
   GP1:
	UF : 1, UT : 1,		CONFIG : 'N U T, 0, 0, 0',
	X =  1646.145  mm,	Y =   -25.939  mm,	Z =   -16.939  mm,
	W =    35.688 deg,	P =    26.418 deg,	R =  -138.451 deg
   GP2:
	UF : 1, UT : 1,
	J1=    90.000 deg,	J2=   -90.000 deg
};
P[663]{
   GP1:
	UF : 1, UT : 1,		CONFIG : 'N U T, 0, 0, 0',
	X =  2051.861  mm,	Y =   -39.046  mm,	Z =    15.590  mm,
	W =    25.849 deg,	P =    22.528 deg,	R =  -155.836 deg
   GP2:
	UF : 1, UT : 1,
	J1=    80.000 deg,	J2=   -90.000 deg
};
P[664]{
   GP1:
	UF : 1, UT : 1,		CONFIG : 'N U T, 0, 0, 1',
	X =  2057.801  mm,	Y =    -3.316  mm,	Z =    14.205  mm,
	W =    26.548 deg,	P =    23.913 deg,	R =  -139.402 deg
   GP2:
	UF : 1, UT : 1,
	J1=    80.000 deg,	J2=   -90.000 deg
};
P[665]{
   GP1:
	UF : 1, UT : 1,		CONFIG : 'N U T, 0, 0, 0',
	X =  2063.971  mm,	Y =     7.752  mm,	Z =    10.705  mm,
	W =    22.379 deg,	P =    28.260 deg,	R =  -174.078 deg
   GP2:
	UF : 1, UT : 1,
	J1=    80.000 deg,	J2=   -90.000 deg
};
P[666]{
   GP1:
	UF : 1, UT : 1,		CONFIG : 'N U T, 0, 0, 0',
	X =  2072.226  mm,	Y =    21.402  mm,	Z =    11.397  mm,
	W =    17.944 deg,	P =    33.020 deg,	R =   153.343 deg
   GP2:
	UF : 1, UT : 1,
	J1=    80.000 deg,	J2=   -90.000 deg
};
P[667]{
   GP1:
	UF : 1, UT : 1,		CONFIG : 'N U T, 0, 0, 0',
	X =  2245.074  mm,	Y =   189.559  mm,	Z =   -20.118  mm,
	W =      .046 deg,	P =    36.124 deg,	R =   125.242 deg
   GP2:
	UF : 1, UT : 1,
	J1=    80.000 deg,	J2=   -90.000 deg
};
P[668]{
   GP1:
	UF : 1, UT : 1,		CONFIG : 'N U T, 0, 0, 0',
	X =  2258.994  mm,	Y =   199.875  mm,	Z =   -22.247  mm,
	W =     3.303 deg,	P =    33.870 deg,	R =   124.421 deg
   GP2:
	UF : 1, UT : 1,
	J1=    80.000 deg,	J2=   -90.000 deg
};
P[669]{
   GP1:
	UF : 1, UT : 1,		CONFIG : 'N U T, 0, 0, 0',
	X =  2274.478  mm,	Y =   212.174  mm,	Z =   -25.111  mm,
	W =     6.003 deg,	P =    35.928 deg,	R =   123.383 deg
   GP2:
	UF : 1, UT : 1,
	J1=    80.000 deg,	J2=   -90.000 deg
};
P[670]{
   GP1:
	UF : 1, UT : 1,		CONFIG : 'N U T, 0, 0, 0',
	X =  2492.536  mm,	Y =   739.403  mm,	Z =    25.184  mm,
	W =   -42.166 deg,	P =     5.515 deg,	R =   107.587 deg
   GP2:
	UF : 1, UT : 1,
	J1=    80.000 deg,	J2=   -90.000 deg
};
P[671]{
   GP1:
	UF : 1, UT : 1,		CONFIG : 'N U T, 0, 0, 0',
	X =  2492.536  mm,	Y =   809.403  mm,	Z =    25.184  mm,
	W =   -38.452 deg,	P =    19.595 deg,	R =   124.425 deg
   GP2:
	UF : 1, UT : 1,
	J1=    80.000 deg,	J2=   -90.000 deg
};
P[672]{
   GP1:
	UF : 1, UT : 1,		CONFIG : 'N U T, 0, 0, 0',
	X =  2372.904  mm,	Y =   273.457  mm,	Z =   -41.545  mm,
	W =     8.789 deg,	P =    37.207 deg,	R =   129.064 deg
   GP2:
	UF : 1, UT : 1,
	J1=    80.000 deg,	J2=   -90.000 deg
};
P[673]{
   GP1:
	UF : 1, UT : 1,		CONFIG : 'N U T, 0, 0, 0',
	X =  2401.399  mm,	Y =   297.467  mm,	Z =   -47.364  mm,
	W =    -2.500 deg,	P =    34.189 deg,	R =   123.664 deg
   GP2:
	UF : 1, UT : 1,
	J1=    80.000 deg,	J2=   -90.000 deg
};
P[674]{
   GP1:
	UF : 1, UT : 1,		CONFIG : 'N U T, 0, 0, 0',
	X =  2407.928  mm,	Y =   304.967  mm,	Z =   -48.330  mm,
	W =      .577 deg,	P =    31.083 deg,	R =   135.857 deg
   GP2:
	UF : 1, UT : 1,
	J1=    80.000 deg,	J2=   -90.000 deg
};
P[675]{
   GP1:
	UF : 1, UT : 1,		CONFIG : 'N U T, 0, 0, 0',
	X =  2491.923  mm,	Y =   422.024  mm,	Z =   -65.101  mm,
	W =   -18.684 deg,	P =    29.858 deg,	R =   100.233 deg
   GP2:
	UF : 1, UT : 1,
	J1=    80.000 deg,	J2=   -90.000 deg
};
P[676]{
   GP1:
	UF : 1, UT : 1,		CONFIG : 'N U T, 0, 0, 0',
	X =  2510.075  mm,	Y =   439.838  mm,	Z =   -66.650  mm,
	W =   -18.818 deg,	P =    32.565 deg,	R =    79.871 deg
   GP2:
	UF : 1, UT : 1,
	J1=    80.000 deg,	J2=   -90.000 deg
};
P[677]{
   GP1:
	UF : 1, UT : 1,		CONFIG : 'N U T, 0, 0, 0',
	X =  2536.078  mm,	Y =   450.433  mm,	Z =   -72.340  mm,
	W =   -17.104 deg,	P =    35.632 deg,	R =    74.627 deg
   GP2:
	UF : 1, UT : 1,
	J1=    80.000 deg,	J2=   -90.000 deg
};
P[678]{
   GP1:
	UF : 1, UT : 1,		CONFIG : 'N U T, 0, 0, 0',
	X =  2563.181  mm,	Y =   457.868  mm,	Z =   -75.386  mm,
	W =   -17.103 deg,	P =    35.627 deg,	R =    74.621 deg
   GP2:
	UF : 1, UT : 1,
	J1=    80.000 deg,	J2=   -90.000 deg
};
P[679]{
   GP1:
	UF : 1, UT : 1,		CONFIG : 'N U T, 0, 0, 0',
	X =  2521.799  mm,	Y =   685.855  mm,	Z =   110.598  mm,
	W =   -11.653 deg,	P =   -32.812 deg,	R =    68.201 deg
   GP2:
	UF : 1, UT : 1,
	J1=    80.000 deg,	J2=   -90.000 deg
};
P[680]{
   GP1:
	UF : 1, UT : 1,		CONFIG : 'N U T, 0, 0, 0',
	X =  2352.111  mm,	Y =   297.878  mm,	Z =   188.758  mm,
	W =   -43.260 deg,	P =    61.542 deg,	R =   123.185 deg
   GP2:
	UF : 1, UT : 1,
	J1=    80.000 deg,	J2=   -90.000 deg
};
P[681]{
   GP1:
	UF : 1, UT : 1,		CONFIG : 'N U T, 0, 0, 0',
	X =  1368.100  mm,	Y =   306.117  mm,	Z =   479.720  mm,
	W =   -19.454 deg,	P =    45.370 deg,	R =   135.446 deg
   GP2:
	UF : 1, UT : 1,
	J1=    80.000 deg,	J2=   -90.000 deg
};
P[682]{
   GP1:
	UF : 1, UT : 1,		CONFIG : 'N U T, 0, 0, 0',
	X =   586.370  mm,	Y =  -785.188  mm,	Z =  2292.509  mm,
	W =   -20.678 deg,	P =   -36.657 deg,	R =     1.573 deg
   GP2:
	UF : 1, UT : 1,
	J1=   180.000 deg,	J2=  -150.000 deg
};
P[683]{
   GP1:
	UF : 1, UT : 1,		CONFIG : 'N U T, 0, 0, 0',
	X =   642.423  mm,	Y = -1094.246  mm,	Z =  1725.795  mm,
